  MoveL 4221 to (-399.34, 339.13, -24.94) mm, rotated rx -180 ry 0 rz 0.01 deg; joints [35.63, -31.489, 74.952, -134.207, 54.383, 150.027]
  MoveL 4222 to (-399.69, 339.08, -24.96) mm, rotated rx 180 ry 0 rz 0.01 deg; joints [35.622, -31.473, 74.919, -134.207, 54.368, 150.017]
  MoveL 4223 to (-400.55, 338.85, -24.99) mm, rotated rx 180 ry 0 rz 0.01 deg; joints [35.6, -31.436, 74.847, -134.212, 54.331, 150]
  MoveL 4224 to (-400.6, 338.83, -24.99) mm, rotated rx -180 ry 0 rz 0.01 deg; joints [35.598, -31.435, 74.844, -134.213, 54.329, 149.999]
  MoveL 4225 to (-401.28, 338.49, -25.02) mm, rotated rx -180 ry 0 rz 0.01 deg; joints [35.577, -31.411, 74.798, -134.224, 54.302, 149.993]
  MoveL 4226 to (-401.4, 338.42, -25.02) mm, rotated rx -180 ry 0 rz 0.01 deg; joints [35.572, -31.407, 74.791, -134.227, 54.298, 149.993]
  MoveL 4227 to (-402.84, 337.05, -25.09) mm, rotated rx -180 ry 0 rz 0.01 deg; joints [35.509, -31.38, 74.742, -134.282, 54.25, 150.013]
  MoveL 4228 to (-402.87, 337.02, -25.09) mm, rotated rx 180 ry 0 rz 0.01 deg; joints [35.508, -31.38, 74.742, -134.284, 54.25, 150.014]
  MoveL 4229 to (-403.75, 334.43, -25.19) mm, rotated rx -180 ry 0 rz 0.01 deg; joints [35.423, -31.422, 74.841, -134.402, 54.245, 150.117]
  MoveL 4230 to (-403.78, 333.95, -25.21) mm, rotated rx 180 ry 0 rz 0.01 deg; joints [35.41, -31.437, 74.874, -134.425, 54.251, 150.141]
  MoveL 4231 to (-403.79, 333.65, -25.22) mm, rotated rx 180 ry 0 rz 0.01 deg; joints [35.402, -31.447, 74.895, -134.439, 54.254, 150.156]
  MoveL 4232 to (-403.79, 333.05, -25.24) mm, rotated rx -180 ry 0 rz 0.01 deg; joints [35.386, -31.467, 74.939, -134.468, 54.263, 150.187]
  MoveL 4233 to (-401.25, 328.08, -25.44) mm, rotated rx -180 ry 0 rz 0.01 deg; joints [35.302, -31.758, 75.562, -134.727, 54.453, 150.531]
  MoveL 4234 to (-395.74, 327.2, -25.64) mm, rotated rx 180 ry 0 rz 0.01 deg; joints [35.383, -32.053, 76.188, -134.809, 54.728, 150.769]
  MoveL 4235 to (-391.79, 331.15, -25.85) mm, rotated rx -180 ry 0 rz 0.01 deg; joints [35.562, -32.103, 76.303, -134.652, 54.865, 150.715]
  MoveL 4236 to (-392.66, 336.66, -26.05) mm, rotated rx 180 ry 0 rz 0.01 deg; joints [35.692, -31.86, 75.812, -134.392, 54.757, 150.418]
  MoveL 4237 to (-397.64, 339.2, -26.25) mm, rotated rx -180 ry 0 rz 0.01 deg; joints [35.664, -31.516, 75.116, -134.241, 54.497, 150.126]
  MoveL 4238 to (-398.51, 339.2, -26.28) mm, rotated rx 180 ry 0 rz 0.01 deg; joints [35.648, -31.472, 75.027, -134.236, 54.457, 150.097]
  MoveL 4239 to (-399.34, 339.13, -26.31) mm, rotated rx 180 ry 0 rz 0.01 deg; joints [35.631, -31.431, 74.946, -134.233, 54.42, 150.072]
  MoveL 4240 to (-399.69, 339.08, -26.32) mm, rotated rx 180 ry 0 rz 0.01 deg; joints [35.622, -31.415, 74.913, -134.233, 54.404, 150.063]
  MoveL 4241 to (-400.55, 338.85, -26.35) mm, rotated rx 180 ry 0 rz 0.01 deg; joints [35.6, -31.379, 74.841, -134.238, 54.368, 150.045]
  MoveL 4242 to (-400.6, 338.83, -26.35) mm, rotated rx 180 ry 0 rz 0.01 deg; joints [35.599, -31.377, 74.838, -134.239, 54.366, 150.045]
  MoveL 4243 to (-401.28, 338.49, -26.38) mm, rotated rx -180 ry 0 rz 0.01 deg; joints [35.577, -31.353, 74.792, -134.25, 54.339, 150.038]
  MoveL 4244 to (-401.4, 338.42, -26.39) mm, rotated rx 180 ry 0 rz 0.01 deg; joints [35.573, -31.35, 74.785, -134.253, 54.334, 150.038]
  MoveL 4245 to (-402.84, 337.05, -26.46) mm, rotated rx -180 ry 0 rz 0.01 deg; joints [35.51, -31.322, 74.737, -134.308, 54.287, 150.059]
  MoveL 4246 to (-402.87, 337.02, -26.46) mm, rotated rx -180 ry 0 rz 0.01 deg; joints [35.509, -31.322, 74.737, -134.31, 54.286, 150.06]
  MoveL 4247 to (-403.75, 334.43, -26.55) mm, rotated rx 180 ry 0 rz 0.01 deg; joints [35.424, -31.364, 74.835, -134.428, 54.282, 150.162]
  MoveL 4248 to (-403.78, 333.95, -26.57) mm, rotated rx -180 ry 0 rz 0.01 deg; joints [35.411, -31.379, 74.868, -134.451, 54.287, 150.186]
  MoveL 4249 to (-403.79, 333.65, -26.58) mm, rotated rx 180 ry 0 rz 0.01 deg; joints [35.403, -31.389, 74.889, -134.465, 54.291, 150.201]
  MoveL 4250 to (-403.79, 333.05, -26.6) mm, rotated rx -180 ry 0 rz 0.01 deg; joints [35.387, -31.409, 74.933, -134.494, 54.3, 150.232]
  MoveL 4251 to (-401.25, 328.08, -26.8) mm, rotated rx 180 ry 0 rz 0.01 deg; joints [35.303, -31.7, 75.556, -134.752, 54.49, 150.576]
  MoveL 4252 to (-395.74, 327.2, -27.01) mm, rotated rx -180 ry 0 rz 0.01 deg; joints [35.384, -31.994, 76.182, -134.834, 54.765, 150.814]
  MoveL 4253 to (-391.79, 331.15, -27.21) mm, rotated rx 180 ry 0 rz 0.01 deg; joints [35.563, -32.044, 76.297, -134.678, 54.902, 150.76]
  MoveL 4254 to (-392.66, 336.66, -27.41) mm, rotated rx 180 ry 0 rz 0.01 deg; joints [35.692, -31.802, 75.806, -134.417, 54.794, 150.464]
  MoveL 4255 to (-397.64, 339.2, -27.61) mm, rotated rx -180 ry 0 rz 0.01 deg; joints [35.665, -31.458, 75.11, -134.267, 54.533, 150.172]
  MoveL 4256 to (-398.51, 339.2, -27.64) mm, rotated rx -180 ry 0 rz 0.01 deg; joints [35.649, -31.414, 75.021, -134.262, 54.494, 150.142]
  MoveL 4257 to (-399.34, 339.13, -27.67) mm, rotated rx -180 ry 0 rz 0.01 deg; joints [35.631, -31.373, 74.94, -134.259, 54.456, 150.117]
  MoveL 4258 to (-399.69, 339.08, -27.69) mm, rotated rx -180 ry 0 rz 0.01 deg; joints [35.623, -31.357, 74.907, -134.259, 54.441, 150.108]
  MoveL 4259 to (-400.55, 338.85, -27.72) mm, rotated rx 180 ry 0 rz 0.01 deg; joints [35.601, -31.321, 74.835, -134.265, 54.404, 150.091]
  MoveL 4260 to (-400.6, 338.83, -27.72) mm, rotated rx -180 ry 0 rz 0.01 deg; joints [35.6, -31.319, 74.832, -134.265, 54.403, 150.09]
  MoveL 4261 to (-401.28, 338.49, -27.75) mm, rotated rx -180 ry 0 rz 0.01 deg; joints [35.578, -31.295, 74.786, -134.276, 54.376, 150.084]
  MoveL 4262 to (-401.4, 338.42, -27.75) mm, rotated rx 180 ry 0 rz 0.01 deg; joints [35.574, -31.292, 74.779, -134.279, 54.371, 150.084]
  MoveL 4263 to (-402.84, 337.05, -27.82) mm, rotated rx -180 ry 0 rz 0.01 deg; joints [35.511, -31.264, 74.731, -134.334, 54.323, 150.104]
  MoveL 4264 to (-402.87, 337.02, -27.82) mm, rotated rx -180 ry 0 rz 0.01 deg; joints [35.509, -31.264, 74.731, -134.336, 54.323, 150.105]
  MoveL 4265 to (-403.75, 334.43, -27.92) mm, rotated rx -180 ry 0 rz 0.01 deg; joints [35.424, -31.307, 74.829, -134.454, 54.318, 150.208]
  MoveL 4266 to (-403.78, 333.95, -27.94) mm, rotated rx -180 ry 0 rz 0.01 deg; joints [35.411, -31.321, 74.862, -134.477, 54.324, 150.232]
  MoveL 4267 to (-403.79, 333.65, -27.95) mm, rotated rx -180 ry 0 rz 0.01 deg; joints [35.403, -31.331, 74.883, -134.491, 54.328, 150.246]
  MoveL 4268 to (-403.79, 333.05, -27.97) mm, rotated rx -180 ry 0 rz 0.01 deg; joints [35.387, -31.351, 74.927, -134.52, 54.336, 150.277]
  MoveL 4269 to (-401.25, 328.08, -28.17) mm, rotated rx -180 ry 0 rz 0.01 deg; joints [35.304, -31.642, 75.55, -134.778, 54.527, 150.621]
  MoveL 4270 to (-395.74, 327.2, -28.37) mm, rotated rx -180 ry 0 rz 0.01 deg; joints [35.384, -31.936, 76.176, -134.86, 54.802, 150.859]
  MoveL 4271 to (-391.79, 331.15, -28.57) mm, rotated rx -180 ry 0 rz 0.01 deg; joints [35.564, -31.986, 76.291, -134.703, 54.939, 150.805]
  MoveL 4272 to (-392.66, 336.66, -28.78) mm, rotated rx -180 ry 0 rz 0.01 deg; joints [35.693, -31.744, 75.8, -134.443, 54.831, 150.509]
  MoveL 4273 to (-397.64, 339.2, -28.98) mm, rotated rx -180 ry 0 rz 0.01 deg; joints [35.666, -31.4, 75.104, -134.293, 54.57, 150.217]
  MoveL 4274 to (-398.51, 339.2, -29.01) mm, rotated rx -180 ry 0 rz 0.01 deg; joints [35.649, -31.356, 75.014, -134.287, 54.53, 150.188]
  MoveL 4275 to (-399.34, 339.13, -29.04) mm, rotated rx -180 ry 0 rz 0.01 deg; joints [35.632, -31.315, 74.934, -134.285, 54.493, 150.163]
  MoveL 4276 to (-399.69, 339.08, -29.05) mm, rotated rx -180 ry 0 rz 0.01 deg; joints [35.624, -31.299, 74.901, -134.285, 54.477, 150.154]
  MoveL 4277 to (-400.55, 338.85, -29.08) mm, rotated rx -180 ry 0 rz 0.01 deg; joints [35.601, -31.263, 74.829, -134.29, 54.441, 150.136]
  MoveL 4278 to (-400.6, 338.83, -29.08) mm, rotated rx -180 ry 0 rz 0.01 deg; joints [35.6, -31.261, 74.826, -134.291, 54.439, 150.135]
  MoveL 4279 to (-401.28, 338.49, -29.11) mm, rotated rx 180 ry 0 rz 0.01 deg; joints [35.578, -31.237, 74.78, -134.302, 54.412, 150.129]
  MoveL 4280 to (-401.4, 338.42, -29.12) mm, rotated rx 180 ry 0 rz 0.01 deg; joints [35.574, -31.234, 74.773, -134.305, 54.407, 150.129]
  MoveL 4281 to (-402.84, 337.05, -29.19) mm, rotated rx -180 ry 0 rz 0.01 deg; joints [35.511, -31.206, 74.724, -134.36, 54.36, 150.149]
  MoveL 4282 to (-402.87, 337.02, -29.19) mm, rotated rx -180 ry 0 rz 0.01 deg; joints [35.51, -31.206, 74.724, -134.362, 54.359, 150.15]
  MoveL 4283 to (-403.75, 334.43, -29.28) mm, rotated rx 180 ry 0 rz 0.01 deg; joints [35.425, -31.248, 74.823, -134.48, 54.355, 150.253]
  MoveL 4284 to (-403.78, 333.95, -29.3) mm, rotated rx -180 ry 0 rz 0.01 deg; joints [35.412, -31.263, 74.856, -134.503, 54.361, 150.277]
  MoveL 4285 to (-403.79, 333.65, -29.31) mm, rotated rx -180 ry 0 rz 0.01 deg; joints [35.404, -31.273, 74.876, -134.517, 54.365, 150.292]
  MoveL 4286 to (-403.79, 333.05, -29.33) mm, rotated rx -180 ry 0 rz 0.01 deg; joints [35.388, -31.293, 74.921, -134.546, 54.373, 150.323]
  MoveL 4287 to (-401.25, 328.08, -29.53) mm, rotated rx -180 ry 0 rz 0.01 deg; joints [35.304, -31.583, 75.544, -134.804, 54.564, 150.666]
  MoveL 4288 to (-395.74, 327.2, -29.74) mm, rotated rx -180 ry 0 rz 0.01 deg; joints [35.385, -31.877, 76.17, -134.885, 54.839, 150.904]
  MoveL 4289 to (-391.79, 331.15, -29.94) mm, rotated rx -180 ry 0 rz 0.01 deg; joints [35.564, -31.927, 76.285, -134.729, 54.976, 150.85]
  MoveL 4290 to (-392.66, 336.66, -30.14) mm, rotated rx -180 ry 0 rz 0.01 deg; joints [35.693, -31.685, 75.794, -134.469, 54.867, 150.554]
  MoveL 4291 to (-397.64, 339.2, -30.34) mm, rotated rx -180 ry 0 rz 0.01 deg; joints [35.666, -31.342, 75.098, -134.319, 54.607, 150.262]
  MoveL 4292 to (-398.51, 339.2, -30.37) mm, rotated rx -180 ry 0 rz 0.01 deg; joints [35.65, -31.297, 75.008, -134.313, 54.567, 150.233]
  MoveL 4293 to (-399.34, 339.13, -30.4) mm, rotated rx -180 ry 0 rz 0.01 deg; joints [35.632, -31.257, 74.927, -134.311, 54.529, 150.208]
  MoveL 4294 to (-399.69, 339.08, -30.42) mm, rotated rx -180 ry 0 rz 0.01 deg; joints [35.624, -31.241, 74.895, -134.311, 54.514, 150.199]
  MoveL 4295 to (-400.55, 338.85, -30.45) mm, rotated rx 180 ry 0 rz 0.01 deg; joints [35.602, -31.204, 74.823, -134.316, 54.477, 150.181]
  MoveL 4296 to (-400.6, 338.83, -30.45) mm, rotated rx 180 ry 0 rz 0.01 deg; joints [35.601, -31.203, 74.819, -134.317, 54.475, 150.18]
  MoveL 4297 to (-401.28, 338.49, -30.47) mm, rotated rx -180 ry 0 rz 0.01 deg; joints [35.579, -31.179, 74.773, -134.328, 54.449, 150.174]
  MoveL 4298 to (-401.4, 338.42, -30.48) mm, rotated rx -180 ry 0 rz 0.01 deg; joints [35.575, -31.175, 74.766, -134.331, 54.444, 150.174]
  MoveL 4299 to (-402.84, 337.05, -30.55) mm, rotated rx -180 ry 0 rz 0.01 deg; joints [35.512, -31.148, 74.718, -134.386, 54.396, 150.194]
  MoveL 4300 to (-402.87, 337.02, -30.55) mm, rotated rx -180 ry 0 rz 0.01 deg; joints [35.51, -31.148, 74.718, -134.388, 54.396, 150.195]
  MoveL 4301 to (-403.75, 334.43, -30.65) mm, rotated rx -180 ry 0 rz 0.01 deg; joints [35.426, -31.19, 74.816, -134.506, 54.391, 150.298]
  MoveL 4302 to (-403.78, 333.95, -30.66) mm, rotated rx 180 ry 0 rz 0.01 deg; joints [35.412, -31.205, 74.849, -134.529, 54.397, 150.322]
  MoveL 4303 to (-403.79, 333.65, -30.68) mm, rotated rx -180 ry 0 rz 0.01 deg; joints [35.405, -31.215, 74.87, -134.543, 54.401, 150.337]
  MoveL 4304 to (-403.79, 333.05, -30.7) mm, rotated rx -180 ry 0 rz 0.01 deg; joints [35.389, -31.235, 74.914, -134.572, 54.41, 150.368]
  MoveL 4305 to (-401.25, 328.08, -30.9) mm, rotated rx 180 ry 0 rz 0.01 deg; joints [35.305, -31.525, 75.538, -134.83, 54.601, 150.711]
  MoveL 4306 to (-395.74, 327.2, -31.1) mm, rotated rx 180 ry 0 rz 0.01 deg; joints [35.385, -31.819, 76.164, -134.911, 54.876, 150.949]
  MoveL 4307 to (-391.79, 331.15, -31.3) mm, rotated rx -180 ry 0 rz 0.01 deg; joints [35.565, -31.869, 76.278, -134.754, 55.013, 150.895]
  MoveL 4308 to (-392.66, 336.66, -31.51) mm, rotated rx 180 ry 0 rz 0.01 deg; joints [35.694, -31.627, 75.787, -134.494, 54.904, 150.599]
  MoveL 4309 to (-397.64, 339.2, -31.71) mm, rotated rx -180 ry 0 rz 0.01 deg; joints [35.667, -31.284, 75.091, -134.345, 54.643, 150.307]
  MoveL 4310 to (-398.51, 339.2, -31.74) mm, rotated rx 180 ry 0 rz 0.01 deg; joints [35.65, -31.239, 75.002, -134.339, 54.603, 150.278]
  MoveL 4311 to (-399.34, 339.13, -31.77) mm, rotated rx 180 ry 0 rz 0.01 deg; joints [35.633, -31.199, 74.921, -134.337, 54.566, 150.253]
  MoveL 4312 to (-399.69, 339.08, -31.78) mm, rotated rx -180 ry 0 rz 0.01 deg; joints [35.625, -31.183, 74.888, -134.337, 54.55, 150.244]
  MoveL 4313 to (-400.55, 338.85, -31.81) mm, rotated rx -180 ry 0 rz 0.01 deg; joints [35.603, -31.146, 74.816, -134.342, 54.514, 150.226]
  MoveL 4314 to (-400.6, 338.83, -31.81) mm, rotated rx -180 ry 0 rz 0.01 deg; joints [35.601, -31.145, 74.813, -134.343, 54.512, 150.225]
  MoveL 4315 to (-401.28, 338.49, -31.84) mm, rotated rx 180 ry 0 rz 0.01 deg; joints [35.58, -31.121, 74.767, -134.354, 54.485, 150.219]
  MoveL 4316 to (-401.4, 338.42, -31.84) mm, rotated rx -180 ry 0 rz 0.01 deg; joints [35.575, -31.117, 74.76, -134.357, 54.48, 150.219]
  MoveL 4317 to (-402.84, 337.05, -31.91) mm, rotated rx -180 ry 0 rz 0.01 deg; joints [35.512, -31.09, 74.711, -134.412, 54.433, 150.239]
  MoveL 4318 to (-402.87, 337.02, -31.92) mm, rotated rx -180 ry 0 rz 0.01 deg; joints [35.511, -31.09, 74.711, -134.414, 54.432, 150.24]
  MoveL 4319 to (-403.75, 334.43, -32.01) mm, rotated rx -180 ry 0 rz 0.01 deg; joints [35.426, -31.132, 74.81, -134.532, 54.428, 150.343]
  MoveL 4320 to (-403.78, 333.95, -32.03) mm, rotated rx -180 ry 0 rz 0.01 deg; joints [35.413, -31.147, 74.843, -134.555, 54.434, 150.367]
  MoveL 4321 to (-403.79, 333.65, -32.04) mm, rotated rx -180 ry 0 rz 0.01 deg; joints [35.405, -31.156, 74.863, -134.569, 54.438, 150.382]
  MoveL 4322 to (-403.79, 333.05, -32.06) mm, rotated rx 180 ry 0 rz 0.01 deg; joints [35.389, -31.177, 74.908, -134.598, 54.446, 150.413]
  MoveL 4323 to (-401.25, 328.08, -32.26) mm, rotated rx 180 ry 0 rz 0.01 deg; joints [35.305, -31.467, 75.531, -134.855, 54.638, 150.756]
  MoveL 4324 to (-395.74, 327.2, -32.47) mm, rotated rx -180 ry 0 rz 0.01 deg; joints [35.386, -31.76, 76.157, -134.936, 54.914, 150.994]
  MoveL 4325 to (-391.79, 331.15, -32.67) mm, rotated rx 180 ry 0 rz 0.01 deg; joints [35.565, -31.81, 76.272, -134.779, 55.05, 150.94]
  MoveL 4326 to (-392.66, 336.66, -32.87) mm, rotated rx -180 ry 0 rz 0.01 deg; joints [35.695, -31.568, 75.781, -134.519, 54.941, 150.644]
  MoveL 4327 to (-397.64, 339.2, -33.07) mm, rotated rx -180 ry 0 rz 0.01 deg; joints [35.667, -31.225, 75.085, -134.37, 54.679, 150.352]
  MoveL 4328 to (-398.51, 339.2, -33.1) mm, rotated rx 180 ry 0 rz 0.01 deg; joints [35.651, -31.181, 74.995, -134.365, 54.639, 150.323]
  MoveL 4329 to (-399.34, 339.13, -33.13) mm, rotated rx -180 ry 0 rz 0.01 deg; joints [35.634, -31.141, 74.914, -134.362, 54.602, 150.298]
  MoveL 4330 to (-399.69, 339.08, -33.14) mm, rotated rx 180 ry 0 rz 0.01 deg; joints [35.625, -31.124, 74.882, -134.363, 54.587, 150.289]
  MoveL 4331 to (-400.55, 338.85, -33.18) mm, rotated rx 180 ry 0 rz 0.01 deg; joints [35.603, -31.088, 74.809, -134.368, 54.55, 150.271]
  MoveL 4332 to (-400.6, 338.83, -33.18) mm, rotated rx -180 ry 0 rz 0.01 deg; joints [35.602, -31.086, 74.806, -134.368, 54.548, 150.27]
  MoveL 4333 to (-401.28, 338.49, -33.2) mm, rotated rx -180 ry 0 rz 0.01 deg; joints [35.58, -31.063, 74.76, -134.38, 54.521, 150.264]
  MoveL 4334 to (-401.4, 338.42, -33.21) mm, rotated rx -180 ry 0 rz 0.01 deg; joints [35.576, -31.059, 74.753, -134.382, 54.517, 150.264]
  MoveL 4335 to (-402.84, 337.05, -33.28) mm, rotated rx 180 ry 0 rz 0.01 deg; joints [35.513, -31.032, 74.705, -134.438, 54.469, 150.284]
  MoveL 4336 to (-402.87, 337.02, -33.28) mm, rotated rx -180 ry 0 rz 0.01 deg; joints [35.512, -31.032, 74.705, -134.439, 54.469, 150.285]
  MoveL 4337 to (-403.75, 334.43, -33.38) mm, rotated rx -180 ry 0 rz 0.01 deg; joints [35.427, -31.074, 74.803, -134.557, 54.464, 150.388]
  MoveL 4338 to (-403.78, 333.95, -33.39) mm, rotated rx -180 ry 0 rz 0.01 deg; joints [35.414, -31.089, 74.836, -134.58, 54.47, 150.411]
  MoveL 4339 to (-403.79, 333.65, -33.4) mm, rotated rx -180 ry 0 rz 0.01 deg; joints [35.406, -31.098, 74.857, -134.594, 54.474, 150.426]
  MoveL 4340 to (-403.79, 333.05, -33.43) mm, rotated rx 180 ry 0 rz 0.01 deg; joints [35.39, -31.118, 74.901, -134.623, 54.483, 150.457]
  MoveL 4341 to (-401.25, 328.08, -33.63) mm, rotated rx -180 ry 0 rz 0.01 deg; joints [35.306, -31.408, 75.525, -134.88, 54.675, 150.8]
  MoveL 4342 to (-395.74, 327.2, -33.83) mm, rotated rx -180 ry 0 rz 0.01 deg; joints [35.387, -31.702, 76.15, -134.961, 54.951, 151.038]
  MoveL 4343 to (-391.79, 331.15, -34.03) mm, rotated rx -180 ry 0 rz 0.01 deg; joints [35.566, -31.751, 76.265, -134.805, 55.087, 150.984]
  MoveL 4344 to (-392.66, 336.66, -34.23) mm, rotated rx 180 ry 0 rz 0.01 deg; joints [35.695, -31.51, 75.774, -134.545, 54.977, 150.689]
  MoveL 4345 to (-397.64, 339.2, -34.44) mm, rotated rx -180 ry 0 rz 0.01 deg; joints [35.668, -31.167, 75.078, -134.396, 54.716, 150.397]
  MoveL 4346 to (-398.51, 339.2, -34.47) mm, rotated rx -180 ry 0 rz 0.01 deg; joints [35.652, -31.122, 74.988, -134.39, 54.676, 150.368]
  MoveL 4347 to (-399.34, 339.13, -34.5) mm, rotated rx 180 ry 0 rz 0.01 deg; joints [35.634, -31.082, 74.907, -134.388, 54.639, 150.343]
  MoveL 4348 to (-399.69, 339.08, -34.51) mm, rotated rx -180 ry 0 rz 0.01 deg; joints [35.626, -31.066, 74.875, -134.388, 54.623, 150.334]
  MoveL 4349 to (-400.55, 338.85, -34.54) mm, rotated rx 180 ry 0 rz 0.01 deg; joints [35.604, -31.03, 74.803, -134.393, 54.586, 150.316]
  MoveL 4350 to (-400.6, 338.83, -34.54) mm, rotated rx 180 ry 0 rz 0.01 deg; joints [35.603, -31.028, 74.799, -134.394, 54.585, 150.315]
  MoveL 4351 to (-401.28, 338.49, -34.57) mm, rotated rx -180 ry 0 rz 0.01 deg; joints [35.581, -31.004, 74.753, -134.405, 54.558, 150.309]
  MoveL 4352 to (-401.4, 338.42, -34.57) mm, rotated rx -180 ry 0 rz 0.01 deg; joints [35.576, -31.001, 74.746, -134.408, 54.553, 150.309]
  MoveL 4353 to (-402.84, 337.05, -34.64) mm, rotated rx -180 ry 0 rz 0.01 deg; joints [35.514, -30.974, 74.698, -134.463, 54.506, 150.329]
  MoveL 4354 to (-402.87, 337.02, -34.64) mm, rotated rx -180 ry 0 rz 0.01 deg; joints [35.512, -30.974, 74.698, -134.465, 54.505, 150.33]
  MoveL 4355 to (-403.75, 334.43, -34.74) mm, rotated rx -180 ry 0 rz 0.01 deg; joints [35.427, -31.015, 74.796, -134.583, 54.501, 150.432]
  MoveL 4356 to (-403.78, 333.95, -34.76) mm, rotated rx -180 ry 0 rz 0.01 deg; joints [35.414, -31.03, 74.829, -134.606, 54.507, 150.456]
  MoveL 4357 to (-403.79, 333.65, -34.77) mm, rotated rx -180 ry 0 rz 0.01 deg; joints [35.406, -31.04, 74.85, -134.62, 54.511, 150.471]
  MoveL 4358 to (-403.79, 333.05, -34.79) mm, rotated rx -180 ry 0 rz 0.01 deg; joints [35.39, -31.06, 74.894, -134.649, 54.519, 150.502]
  MoveL 4359 to (-401.25, 328.08, -34.99) mm, rotated rx -180 ry 0 rz 0.01 deg; joints [35.307, -31.35, 75.518, -134.906, 54.712, 150.845]
  MoveL 4360 to (-395.74, 327.2, -35.19) mm, rotated rx 180 ry 0 rz 0.01 deg; joints [35.387, -31.643, 76.144, -134.986, 54.988, 151.083]
  MoveL 4361 to (-391.79, 331.15, -35.4) mm, rotated rx 180 ry 0 rz 0.01 deg; joints [35.566, -31.692, 76.258, -134.83, 55.124, 151.029]
  MoveL 4362 to (-392.66, 336.66, -35.6) mm, rotated rx 180 ry 0 rz 0.01 deg; joints [35.696, -31.451, 75.767, -134.57, 55.014, 150.733]
  MoveL 4363 to (-397.64, 339.2, -35.8) mm, rotated rx 180 ry 0 rz 0.01 deg; joints [35.669, -31.108, 75.071, -134.421, 54.752, 150.442]
  MoveL 4364 to (-398.51, 339.2, -35.83) mm, rotated rx -180 ry 0 rz 0.01 deg; joints [35.652, -31.064, 74.981, -134.416, 54.712, 150.412]
  MoveL 4365 to (-399.34, 339.13, -35.86) mm, rotated rx -180 ry 0 rz 0.01 deg; joints [35.635, -31.024, 74.9, -134.413, 54.675, 150.387]
  MoveL 4366 to (-399.69, 339.08, -35.87) mm, rotated rx -180 ry 0 rz 0.01 deg; joints [35.627, -31.007, 74.868, -134.414, 54.659, 150.378]
  MoveL 4367 to (-400.55, 338.85, -35.9) mm, rotated rx -180 ry 0 rz 0.01 deg; joints [35.604, -30.971, 74.796, -134.419, 54.623, 150.361]
  MoveL 4368 to (-400.6, 338.83, -35.91) mm, rotated rx -180 ry 0 rz 0.01 deg; joints [35.603, -30.97, 74.792, -134.419, 54.621, 150.36]
  MoveL 4369 to (-401.28, 338.49, -35.93) mm, rotated rx -180 ry 0 rz 0.01 deg; joints [35.581, -30.946, 74.746, -134.431, 54.594, 150.354]
  MoveL 4370 to (-401.4, 338.42, -35.94) mm, rotated rx -180 ry 0 rz 0.01 deg; joints [35.577, -30.942, 74.739, -134.434, 54.589, 150.353]
  MoveL 4371 to (-402.84, 337.05, -36.01) mm, rotated rx -180 ry 0 rz 0.01 deg; joints [35.514, -30.915, 74.691, -134.489, 54.542, 150.374]
  MoveL 4372 to (-402.87, 337.02, -36.01) mm, rotated rx -180 ry 0 rz 0.01 deg; joints [35.513, -30.915, 74.691, -134.49, 54.541, 150.375]
  MoveL 4373 to (-403.75, 334.43, -36.11) mm, rotated rx -180 ry 0 rz 0.01 deg; joints [35.428, -30.957, 74.789, -134.608, 54.537, 150.477]
  MoveL 4374 to (-403.78, 333.95, -36.12) mm, rotated rx -180 ry 0 rz 0.01 deg; joints [35.415, -30.972, 74.822, -134.631, 54.543, 150.501]
  MoveL 4375 to (-403.79, 333.65, -36.13) mm, rotated rx -180 ry 0 rz 0.01 deg; joints [35.407, -30.981, 74.843, -134.645, 54.547, 150.516]
  MoveL 4376 to (-403.79, 333.05, -36.15) mm, rotated rx -180 ry 0 rz 0.01 deg; joints [35.391, -31.001, 74.887, -134.674, 54.556, 150.546]
  MoveL 4377 to (-401.25, 328.08, -36.36) mm, rotated rx -180 ry 0 rz 0.01 deg; joints [35.307, -31.291, 75.511, -134.931, 54.749, 150.889]
  MoveL 4378 to (-395.74, 327.2, -36.56) mm, rotated rx 180 ry 0 rz 0.01 deg; joints [35.388, -31.584, 76.137, -135.012, 55.025, 151.127]
  MoveL 4379 to (-391.79, 331.15, -36.76) mm, rotated rx -180 ry 0 rz 0.01 deg; joints [35.567, -31.634, 76.251, -134.855, 55.161, 151.073]
  MoveL 4380 to (-392.66, 336.66, -36.96) mm, rotated rx 180 ry 0 rz 0.01 deg; joints [35.696, -31.392, 75.76, -134.595, 55.051, 150.778]
  MoveL 4381 to (-397.64, 339.2, -37.17) mm, rotated rx -180 ry 0 rz 0.01 deg; joints [35.669, -31.05, 75.064, -134.446, 54.788, 150.486]
  MoveL 4382 to (-398.51, 339.2, -37.2) mm, rotated rx -180 ry 0 rz 0.01 deg; joints [35.653, -31.005, 74.974, -134.441, 54.748, 150.457]
  MoveL 4383 to (-399.34, 339.13, -37.23) mm, rotated rx -180 ry 0 rz 0.01 deg; joints [35.635, -30.965, 74.893, -134.439, 54.711, 150.432]
  MoveL 4384 to (-399.69, 339.08, -37.24) mm, rotated rx -180 ry 0 rz 0.01 deg; joints [35.627, -30.949, 74.861, -134.439, 54.695, 150.423]
  MoveL 4385 to (-400.55, 338.85, -37.27) mm, rotated rx 180 ry 0 rz 0.01 deg; joints [35.605, -30.913, 74.788, -134.444, 54.659, 150.405]
  MoveL 4386 to (-400.6, 338.83, -37.27) mm, rotated rx -180 ry 0 rz 0.01 deg; joints [35.604, -30.911, 74.785, -134.445, 54.657, 150.404]
  MoveL 4387 to (-401.28, 338.49, -37.3) mm, rotated rx 180 ry 0 rz 0.01 deg; joints [35.582, -30.888, 74.739, -134.456, 54.63, 150.398]
  MoveL 4388 to (-401.4, 338.42, -37.3) mm, rotated rx -180 ry 0 rz 0.01 deg; joints [35.578, -30.884, 74.732, -134.459, 54.625, 150.398]
  MoveL 4389 to (-402.84, 337.05, -37.37) mm, rotated rx -180 ry 0 rz 0.01 deg; joints [35.515, -30.857, 74.684, -134.514, 54.578, 150.418]
  MoveL 4390 to (-402.87, 337.02, -37.37) mm, rotated rx -180 ry 0 rz 0.01 deg; joints [35.513, -30.857, 74.684, -134.516, 54.578, 150.419]
  MoveL 4391 to (-403.75, 334.43, -37.47) mm, rotated rx 180 ry 0 rz 0.01 deg; joints [35.429, -30.899, 74.782, -134.634, 54.574, 150.521]
  MoveL 4392 to (-403.78, 333.95, -37.49) mm, rotated rx -180 ry 0 rz 0.01 deg; joints [35.415, -30.913, 74.815, -134.657, 54.58, 150.545]
  MoveL 4393 to (-403.79, 333.65, -37.5) mm, rotated rx 180 ry 0 rz 0.01 deg; joints [35.407, -30.923, 74.836, -134.671, 54.583, 150.56]
  MoveL 4394 to (-403.79, 333.05, -37.52) mm, rotated rx 180 ry 0 rz 0.01 deg; joints [35.392, -30.943, 74.88, -134.7, 54.592, 150.591]
  MoveL 4395 to (-401.25, 328.08, -37.72) mm, rotated rx -180 ry 0 rz 0.01 deg; joints [35.308, -31.232, 75.503, -134.956, 54.785, 150.934]
  MoveL 4396 to (-395.74, 327.2, -37.92) mm, rotated rx 180 ry 0 rz 0.01 deg; joints [35.388, -31.525, 76.129, -135.036, 55.061, 151.172]
  MoveL 4397 to (-391.79, 331.15, -38.13) mm, rotated rx -180 ry 0 rz 0.01 deg; joints [35.568, -31.575, 76.244, -134.88, 55.198, 151.118]
  MoveL 4398 to (-392.66, 336.66, -38.33) mm, rotated rx -180 ry 0 rz 0.01 deg; joints [35.697, -31.333, 75.753, -134.62, 55.087, 150.822]
  MoveL 4399 to (-397.64, 339.2, -38.53) mm, rotated rx -180 ry 0 rz 0.01 deg; joints [35.67, -30.991, 75.056, -134.472, 54.825, 150.531]
  MoveL 4400 to (-398.51, 339.2, -38.56) mm, rotated rx -180 ry 0 rz 0.01 deg; joints [35.653, -30.947, 74.967, -134.466, 54.785, 150.501]
  MoveL 4401 to (-399.34, 339.13, -38.59) mm, rotated rx -180 ry 0 rz 0.01 deg; joints [35.636, -30.907, 74.886, -134.464, 54.747, 150.476]
  MoveL 4402 to (-399.69, 339.08, -38.6) mm, rotated rx 180 ry 0 rz 0.01 deg; joints [35.628, -30.89, 74.853, -134.464, 54.732, 150.467]
  MoveL 4403 to (-400.55, 338.85, -38.63) mm, rotated rx 180 ry 0 rz 0.01 deg; joints [35.606, -30.854, 74.781, -134.469, 54.695, 150.45]
  MoveL 4404 to (-400.6, 338.83, -38.64) mm, rotated rx -180 ry 0 rz 0.01 deg; joints [35.604, -30.852, 74.778, -134.47, 54.693, 150.449]
  MoveL 4405 to (-401.28, 338.49, -38.66) mm, rotated rx -180 ry 0 rz 0.01 deg; joints [35.583, -30.829, 74.732, -134.481, 54.666, 150.443]
  MoveL 4406 to (-401.4, 338.42, -38.67) mm, rotated rx -180 ry 0 rz 0.01 deg; joints [35.578, -30.825, 74.725, -134.484, 54.662, 150.442]
  MoveL 4407 to (-402.84, 337.05, -38.74) mm, rotated rx -180 ry 0 rz 0.01 deg; joints [35.515, -30.798, 74.676, -134.54, 54.614, 150.463]
  MoveL 4408 to (-402.87, 337.02, -38.74) mm, rotated rx -180 ry 0 rz 0.01 deg; joints [35.514, -30.798, 74.676, -134.541, 54.614, 150.464]
  MoveL 4409 to (-403.75, 334.43, -38.84) mm, rotated rx -180 ry 0 rz 0.01 deg; joints [35.429, -30.84, 74.775, -134.659, 54.61, 150.566]
  MoveL 4410 to (-403.78, 333.95, -38.85) mm, rotated rx -180 ry 0 rz 0.01 deg; joints [35.416, -30.855, 74.807, -134.682, 54.616, 150.59]
  MoveL 4411 to (-403.79, 333.65, -38.86) mm, rotated rx -180 ry 0 rz 0.01 deg; joints [35.408, -30.864, 74.828, -134.696, 54.62, 150.604]
  MoveL 4412 to (-403.79, 333.05, -38.88) mm, rotated rx -180 ry 0 rz 0.01 deg; joints [35.392, -30.884, 74.872, -134.725, 54.629, 150.635]
  MoveL 4413 to (-401.25, 328.08, -39.09) mm, rotated rx 180 ry 0 rz 0.01 deg; joints [35.308, -31.173, 75.496, -134.981, 54.822, 150.978]
  MoveL 4414 to (-395.74, 327.2, -39.29) mm, rotated rx -180 ry 0 rz 0.01 deg; joints [35.389, -31.466, 76.122, -135.061, 55.098, 151.216]
  MoveL 4415 to (-391.79, 331.15, -39.49) mm, rotated rx -180 ry 0 rz 0.01 deg; joints [35.568, -31.516, 76.236, -134.904, 55.234, 151.162]
  MoveL 4416 to (-392.66, 336.66, -39.69) mm, rotated rx 180 ry 0 rz 0.01 deg; joints [35.698, -31.274, 75.745, -134.645, 55.124, 150.867]
  MoveL 4417 to (-397.64, 339.2, -39.9) mm, rotated rx -180 ry 0 rz 0.01 deg; joints [35.67, -30.932, 75.049, -134.497, 54.861, 150.575]
  MoveL 4418 to (-398.51, 339.2, -39.93) mm, rotated rx -180 ry 0 rz 0.01 deg; joints [35.654, -30.888, 74.959, -134.491, 54.821, 150.546]
  MoveL 4419 to (-399.34, 339.13, -39.95) mm, rotated rx -180 ry 0 rz 0.01 deg; joints [35.637, -30.848, 74.878, -134.489, 54.783, 150.521]
  MoveL 4420 to (-399.69, 339.08, -39.97) mm, rotated rx -180 ry 0 rz 0.01 deg; joints [35.628, -30.832, 74.846, -134.489, 54.768, 150.512]
  MoveL 4421 to (-400.55, 338.85, -40) mm, rotated rx -180 ry 0 rz 0.01 deg; joints [35.606, -30.795, 74.774, -134.495, 54.731, 150.494]
  MoveL 4422 to (-400.6, 338.83, -40) mm, rotated rx -180 ry 0 rz 0.01 deg; joints [35.605, -30.794, 74.77, -134.495, 54.729, 150.493]
  MoveL 4423 to (-400.13, 339.01, -40) mm, rotated rx -180 ry 0 rz 0.01 deg; joints [35.618, -30.811, 74.805, -134.49, 54.749, 150.501]
  MoveL 4424 to (-398.92, 339.2, -40) mm, rotated rx -180 ry 0 rz 0.01 deg; joints [35.646, -30.864, 74.916, -134.49, 54.803, 150.533]
  MoveL 4425 to (-213.35, 339.2, -40) mm, rotated rx 180 ry 0 rz 0.01 deg; joints [39.468, -38.9, 91.717, -134.344, 62.753, 155.77]
  MoveL 4426 to (-213.55, 339.16, -40) mm, rotated rx 180 ry 0 rz 0.01 deg; joints [39.462, -38.894, 91.704, -134.347, 62.746, 155.767]
  MoveL 4427 to (-214.63, 338.89, -40) mm, rotated rx 180 ry 0 rz 0.01 deg; joints [39.43, -38.861, 91.635, -134.366, 62.707, 155.753]
  MoveL 4428 to (-215.28, 338.65, -40) mm, rotated rx 180 ry 0 rz 0.01 deg; joints [39.409, -38.844, 91.598, -134.38, 62.685, 155.748]
  MoveL 4429 to (-225.8, 333.55, -40) mm, rotated rx -180 ry 0 rz 0.01 deg; joints [39.036, -38.596, 91.083, -134.661, 62.336, 155.712]
  MoveL 4430 to (-226.11, 333.38, -40) mm, rotated rx 180 ry 0 rz 0.01 deg; joints [39.024, -38.589, 91.069, -134.67, 62.326, 155.712]
  MoveL 4431 to (-227.57, 332.48, -40) mm, rotated rx 180 ry 0 rz 0.01 deg; joints [38.967, -38.56, 91.01, -134.716, 62.28, 155.715]
  MoveL 4432 to (-228.07, 332.1, -40) mm, rotated rx 180 ry 0 rz 0.01 deg; joints [38.946, -38.553, 90.994, -134.735, 62.265, 155.719]
  MoveL 4433 to (-229.52, 330.77, -40) mm, rotated rx -180 ry 0 rz 0.01 deg; joints [38.877, -38.537, 90.964, -134.799, 62.224, 155.74]
  MoveL 4434 to (-229.56, 330.73, -40) mm, rotated rx 180 ry 0 rz 0.01 deg; joints [38.875, -38.537, 90.963, -134.801, 62.223, 155.741]
  MoveL 4435 to (-236.64, 324.01, -40) mm, rotated rx 180 ry 0 rz 0.01 deg; joints [38.536, -38.466, 90.823, -135.122, 62.028, 155.852]
  MoveL 4436 to (-236.94, 323.69, -40) mm, rotated rx 180 ry 0 rz 0.01 deg; joints [38.52, -38.464, 90.82, -135.137, 62.02, 155.858]
  MoveL 4437 to (-237.82, 322.6, -40) mm, rotated rx -180 ry 0 rz 0.01 deg; joints [38.471, -38.463, 90.818, -135.187, 61.999, 155.882]
  MoveL 4438 to (-238.12, 322.17, -40) mm, rotated rx -180 ry 0 rz 0.01 deg; joints [38.453, -38.464, 90.822, -135.207, 61.993, 155.893]
  MoveL 4439 to (-240.45, 318.18, -40) mm, rotated rx -180 ry 0 rz 0.01 deg; joints [38.292, -38.493, 90.89, -135.386, 61.951, 156.002]
  MoveL 4440 to (-240.49, 318.11, -40) mm, rotated rx 180 ry 0 rz 0.01 deg; joints [38.289, -38.494, 90.891, -135.389, 61.95, 156.005]
  MoveL 4441 to (-243.68, 312.3, -40) mm, rotated rx -180 ry 0 rz 0.01 deg; joints [38.059, -38.544, 91.004, -135.648, 61.897, 156.168]
  MoveL 4442 to (-243.84, 311.95, -40) mm, rotated rx 180 ry 0 rz 0.01 deg; joints [38.046, -38.548, 91.013, -135.663, 61.895, 156.178]
  MoveL 4443 to (-244.73, 309.78, -40) mm, rotated rx 180 ry 0 rz 0.01 deg; joints [37.967, -38.578, 91.08, -135.759, 61.888, 156.247]
  MoveL 4444 to (-244.95, 309.01, -40) mm, rotated rx -180 ry 0 rz 0.01 deg; joints [37.941, -38.592, 91.111, -135.792, 61.889, 156.273]
  MoveL 4445 to (-246.39, 299.58, -40) mm, rotated rx 180 ry 0 rz 0.01 deg; joints [37.647, -38.815, 91.595, -136.19, 61.953, 156.624]
  MoveL 4446 to (-246.42, 299.36, -40) mm, rotated rx 180 ry 0 rz 0.01 deg; joints [37.64, -38.821, 91.607, -136.2, 61.955, 156.632]
  MoveL 4447 to (-246.51, 298.27, -40) mm, rotated rx -180 ry 0 rz 0.01 deg; joints [37.608, -38.849, 91.669, -136.245, 61.965, 156.674]
  MoveC 4448 to (-246.51, 297.75, -40) mm, rotated rx -180 ry 0 rz 0.01 deg; joints [37.593, -38.864, 91.701, -136.267, 61.972, 156.695] to (-246.44, 297.24, -40) mm, rotated rx -180 ry 0 rz 0.01 deg; joints [37.581, -38.882, 91.739, -136.287, 61.981, 156.718]
  MoveL 4449 to (-245.04, 290.98, -40) mm, rotated rx 180 ry 0 rz 0.01 deg; joints [37.435, -39.119, 92.249, -136.537, 62.118, 157.002]
  MoveL 4450 to (-245.03, 290.91, -40) mm, rotated rx 180 ry 0 rz 0.01 deg; joints [37.434, -39.122, 92.255, -136.54, 62.12, 157.005]
  MoveL 4451 to (-244.07, 287.02, -40) mm, rotated rx 180 ry 0 rz 0.01 deg; joints [37.344, -39.272, 92.578, -136.694, 62.209, 157.183]
  MoveL 4452 to (-243.75, 286.18, -40) mm, rotated rx 180 ry 0 rz 0.01 deg; joints [37.328, -39.308, 92.656, -136.726, 62.232, 157.224]
  MoveL 4453 to (-241.42, 281.98, -40) mm, rotated rx -180 ry 0 rz 0.01 deg; joints [37.259, -39.519, 93.108, -136.884, 62.38, 157.444]
  MoveL 4454 to (-241.22, 281.66, -40) mm, rotated rx -180 ry 0 rz 0.01 deg; joints [37.254, -39.536, 93.144, -136.896, 62.392, 157.461]
  MoveL 4455 to (-240.29, 280.35, -40) mm, rotated rx 180 ry 0 rz 0.01 deg; joints [37.237, -39.609, 93.301, -136.943, 62.446, 157.534]
  MoveL 4456 to (-240.11, 280.11, -40) mm, rotated rx -180 ry 0 rz 0.01 deg; joints [37.234, -39.623, 93.331, -136.952, 62.457, 157.548]
  MoveL 4457 to (-237.06, 276.55, -40) mm, rotated rx 180 ry 0 rz 0.01 deg; joints [37.199, -39.842, 93.798, -137.077, 62.625, 157.756]
  MoveL 4458 to (-236.75, 276.23, -40) mm, rotated rx 180 ry 0 rz 0.01 deg; joints [37.197, -39.863, 93.844, -137.087, 62.641, 157.776]
  MoveL 4459 to (-236.39, 275.91, -40) mm, rotated rx 180 ry 0 rz 0.01 deg; joints [37.195, -39.886, 93.893, -137.098, 62.66, 157.797]
  MoveL 4460 to (-236.12, 275.69, -40) mm, rotated rx -180 ry 0 rz 0.01 deg; joints [37.195, -39.903, 93.928, -137.105, 62.674, 157.811]
  MoveL 4461 to (-230.67, 271.73, -40) mm, rotated rx -180 ry 0 rz 0.01 deg; joints [37.2, -40.222, 94.611, -137.227, 62.942, 158.086]
  MoveL 4462 to (-230.2, 271.44, -40) mm, rotated rx 180 ry 0 rz 0.01 deg; joints [37.202, -40.248, 94.667, -137.235, 62.965, 158.108]
  MoveL 4463 to (-227.17, 269.92, -40) mm, rotated rx -180 ry 0 rz 0.01 deg; joints [37.224, -40.406, 95.003, -137.274, 63.104, 158.233]
  MoveL 4464 to (-226.74, 269.75, -40) mm, rotated rx 180 ry 0 rz 0.01 deg; joints [37.228, -40.427, 95.048, -137.277, 63.124, 158.249]
  MoveL 4465 to (-223.24, 268.55, -40) mm, rotated rx 180 ry 0 rz 0.01 deg; joints [37.271, -40.592, 95.401, -137.298, 63.278, 158.371]
  MoveL 4466 to (-222.62, 268.41, -40) mm, rotated rx -180 ry 0 rz 0.01 deg; joints [37.28, -40.62, 95.459, -137.299, 63.304, 158.391]
  MoveL 4467 to (-215.36, 267.4, -40) mm, rotated rx -180 ry 0 rz 0.01 deg; joints [37.41, -40.92, 96.098, -137.279, 63.603, 158.586]
  MoveL 4468 to (-214.9, 267.36, -40) mm, rotated rx -180 ry 0 rz 0.01 deg; joints [37.42, -40.939, 96.136, -137.277, 63.622, 158.597]
  MoveL 4469 to (-178.62, 267.36, -40) mm, rotated rx -180 ry 0 rz 0.01 deg; joints [38.234, -42.265, 98.956, -136.93, 65.027, 159.354]
  MoveL 4470 to (-178.15, 267.4, -40) mm, rotated rx -180 ry 0 rz 0.01 deg; joints [38.246, -42.28, 98.99, -136.924, 65.044, 159.362]
  MoveL 4471 to (-170.89, 268.41, -40) mm, rotated rx 180 ry 0 rz 0.01 deg; joints [38.442, -42.511, 99.481, -136.806, 65.307, 159.472]
  MoveL 4472 to (-170.31, 268.54, -40) mm, rotated rx 180 ry 0 rz 0.01 deg; joints [38.459, -42.528, 99.517, -136.794, 65.327, 159.479]
  MoveL 4473 to (-167.48, 269.46, -40) mm, rotated rx -180 ry 0 rz 0.01 deg; joints [38.551, -42.604, 99.676, -136.726, 65.423, 159.502]
  MoveL 4474 to (-167.1, 269.61, -40) mm, rotated rx -180 ry 0 rz 0.01 deg; joints [38.564, -42.613, 99.695, -136.716, 65.435, 159.504]
  MoveL 4475 to (-164.14, 270.98, -40) mm, rotated rx 180 ry 0 rz 0.01 deg; joints [38.673, -42.68, 99.836, -136.629, 65.529, 159.512]
  MoveL 4476 to (-163.71, 271.21, -40) mm, rotated rx -180 ry 0 rz 0.01 deg; joints [38.689, -42.688, 99.854, -136.614, 65.542, 159.512]
  MoveL 4477 to (-161.53, 272.63, -40) mm, rotated rx 180 ry 0 rz 0.01 deg; joints [38.781, -42.726, 99.932, -136.534, 65.606, 159.503]
  MoveL 4478 to (-161.34, 272.76, -40) mm, rotated rx 180 ry 0 rz 0.01 deg; joints [38.79, -42.729, 99.939, -136.526, 65.611, 159.502]
  MoveL 4479 to (-156.98, 276.05, -40) mm, rotated rx -180 ry 0 rz 0.01 deg; joints [38.987, -42.792, 100.067, -136.346, 65.733, 159.467]
  MoveL 4480 to (-156.45, 276.55, -40) mm, rotated rx -180 ry 0 rz 0.01 deg; joints [39.014, -42.797, 100.077, -136.32, 65.746, 159.459]
  MoveL 4481 to (-153.97, 279.45, -40) mm, rotated rx -180 ry 0 rz 0.01 deg; joints [39.156, -42.803, 100.086, -136.176, 65.801, 159.4]
  MoveL 4482 to (-153.84, 279.61, -40) mm, rotated rx 180 ry 0 rz 0.01 deg; joints [39.163, -42.803, 100.086, -136.169, 65.804, 159.397]
  MoveL 4483 to (-152.35, 281.58, -40) mm, rotated rx -180 ry 0 rz 0.01 deg; joints [39.255, -42.801, 100.078, -136.074, 65.834, 159.353]
  MoveL 4484 to (-152.09, 281.98, -40) mm, rotated rx 180 ry 0 rz 0.01 deg; joints [39.273, -42.799, 100.073, -136.055, 65.839, 159.343]
  MoveL 4485 to (-149.77, 286.18, -40) mm, rotated rx -180 ry 0 rz 0.01 deg; joints [39.449, -42.763, 99.989, -135.861, 65.871, 159.232]
  MoveL 4486 to (-149.43, 287.04, -40) mm, rotated rx -180 ry 0 rz 0.01 deg; joints [39.481, -42.751, 99.962, -135.824, 65.872, 159.207]
  MoveL 4487 to (-147.12, 296.84, -40) mm, rotated rx 180 ry 0 rz 0.01 deg; joints [39.816, -42.556, 99.532, -135.41, 65.831, 158.884]
  MoveL 4488 to (-147.03, 297.46, -40) mm, rotated rx -180 ry 0 rz 0.01 deg; joints [39.836, -42.542, 99.5, -135.385, 65.826, 158.862]
  MoveL 4489 to (-146.99, 298.18, -40) mm, rotated rx 180 ry 0 rz 0.01 deg; joints [39.857, -42.522, 99.457, -135.356, 65.818, 158.835]
  MoveL 4490 to (-147.03, 298.84, -40) mm, rotated rx 180 ry 0 rz 0.01 deg; joints [39.875, -42.503, 99.414, -135.33, 65.808, 158.81]
  MoveL 4491 to (-148.48, 308.63, -40) mm, rotated rx 180 ry 0 rz 0.01 deg; joints [40.118, -42.172, 98.696, -134.961, 65.627, 158.405]
  MoveL 4492 to (-148.63, 309.24, -40) mm, rotated rx 180 ry 0 rz 0.01 deg; joints [40.132, -42.15, 98.647, -134.939, 65.613, 158.379]
  MoveL 4493 to (-149.26, 311.05, -40) mm, rotated rx 180 ry 0 rz 0.01 deg; joints [40.168, -42.076, 98.486, -134.874, 65.567, 158.296]
  MoveL 4494 to (-149.46, 311.52, -40) mm, rotated rx 180 ry 0 rz 0.01 deg; joints [40.176, -42.055, 98.441, -134.858, 65.553, 158.274]
  MoveL 4495 to (-151.37, 315.15, -40) mm, rotated rx -180 ry 0 rz 0.01 deg; joints [40.233, -41.883, 98.07, -134.736, 65.435, 158.094]
  MoveL 4496 to (-151.42, 315.25, -40) mm, rotated rx -180 ry 0 rz 0.01 deg; joints [40.234, -41.879, 98.06, -134.733, 65.432, 158.089]
  MoveL 4497 to (-155.13, 321.78, -40) mm, rotated rx 180 ry 0 rz 0.01 deg; joints [40.329, -41.558, 97.368, -134.516, 65.208, 157.758]
  MoveL 4498 to (-155.37, 322.14, -40) mm, rotated rx 180 ry 0 rz 0.01 deg; joints [40.333, -41.539, 97.327, -134.504, 65.195, 157.738]
  MoveL 4499 to (-156.19, 323.23, -40) mm, rotated rx -180 ry 0 rz 0.01 deg; joints [40.344, -41.478, 97.196, -134.47, 65.15, 157.678]
  MoveL 4500 to (-156.47, 323.55, -40) mm, rotated rx 180 ry 0 rz 0.01 deg; joints [40.347, -41.458, 97.154, -134.46, 65.135, 157.66]
  MoveL 4501 to (-157.53, 324.64, -40) mm, rotated rx 180 ry 0 rz 0.01 deg; joints [40.352, -41.389, 97.005, -134.429, 65.081, 157.595]
  MoveL 4502 to (-157.63, 324.74, -40) mm, rotated rx 180 ry 0 rz 0.01 deg; joints [40.352, -41.382, 96.991, -134.426, 65.076, 157.589]
  MoveL 4503 to (-165.05, 331.75, -40) mm, rotated rx 180 ry 0 rz 0.01 deg; joints [40.372, -40.91, 95.979, -134.225, 64.707, 157.153]
  MoveL 4504 to (-165.4, 332.04, -40) mm, rotated rx 180 ry 0 rz 0.01 deg; joints [40.372, -40.889, 95.933, -134.217, 64.69, 157.134]
  MoveL 4505 to (-166.85, 333.08, -40) mm, rotated rx 180 ry 0 rz 0.01 deg; joints [40.366, -40.806, 95.755, -134.19, 64.622, 157.062]
  MoveL 4506 to (-167.34, 333.37, -40) mm, rotated rx -180 ry 0 rz 0.01 deg; joints [40.363, -40.78, 95.699, -134.184, 64.599, 157.039]
  MoveL 4507 to (-177.86, 338.5, -40) mm, rotated rx 180 ry 0 rz 0.01 deg; joints [40.258, -40.245, 94.558, -134.08, 64.134, 156.604]
  MoveL 4508 to (-178.19, 338.64, -40) mm, rotated rx -180 ry 0 rz 0.01 deg; joints [40.255, -40.228, 94.524, -134.078, 64.12, 156.591]
  MoveL 4509 to (-178.91, 338.9, -40) mm, rotated rx 180 ry 0 rz 0.01 deg; joints [40.245, -40.194, 94.451, -134.074, 64.089, 156.564]
  MoveL 4510 to (-179.55, 339.06, -40) mm, rotated rx 180 ry 0 rz 0.01 deg; joints [40.235, -40.166, 94.391, -134.073, 64.062, 156.543]
  MoveL 4511 to (-180.46, 339.2, -40) mm, rotated rx 180 ry 0 rz 0.01 deg; joints [40.218, -40.128, 94.311, -134.076, 64.026, 156.518]
  MoveL 4512 to (4.87, 339.21, -40) mm, rotated rx -180 ry 0 rz 0.01 deg; joints [44.916, -46.237, 107.372, -131.517, 70.593, 160.189]
  MoveL 4513 to (5.94, 339.15, -40) mm, rotated rx -180 ry 0 rz 0.01 deg; joints [44.944, -46.27, 107.444, -131.5, 70.629, 160.211]
  MoveL 4514 to (6.8, 338.95, -40) mm, rotated rx 180 ry 0 rz 0.01 deg; joints [44.963, -46.301, 107.512, -131.491, 70.66, 160.233]
  MoveL 4515 to (7.07, 338.84, -40) mm, rotated rx 180 ry 0 rz 0.01 deg; joints [44.967, -46.313, 107.537, -131.49, 70.671, 160.243]
  MoveL 4516 to (7.37, 338.63, -40) mm, rotated rx 180 ry 0 rz 0.01 deg; joints [44.97, -46.328, 107.569, -131.492, 70.683, 160.256]
  MoveL 4517 to (9.66, 336.38, -40) mm, rotated rx -180 ry 0 rz 0.01 deg; joints [44.971, -46.46, 107.86, -131.533, 70.788, 160.381]
  MoveL 4518 to (9.9, 336.02, -40) mm, rotated rx 180 ry 0 rz 0.01 deg; joints [44.967, -46.477, 107.898, -131.542, 70.801, 160.398]
  MoveL 4519 to (10.07, 335.56, -40) mm, rotated rx -180 ry 0 rz 0.01 deg; joints [44.959, -46.496, 107.938, -131.555, 70.813, 160.418]
  MoveL 4520 to (10.27, 334.35, -40) mm, rotated rx -180 ry 0 rz 0.01 deg; joints [44.931, -46.536, 108.028, -131.596, 70.835, 160.467]
  MoveL 4521 to (10.27, 31.87, -40) mm, rotated rx 180 ry 0 rz 0.01 deg; joints [35.133, -53.75, 124.619, -143.431, 75.064, 170.12]
  MoveL 4522 to (9.18, 36.46, -40) mm, rotated rx 180 ry 0 rz 0.01 deg; joints [35.275, -53.63, 124.332, -143.261, 74.958, 169.978]
  MoveL 4523 to (9.03, 36.92, -40) mm, rotated rx 180 ry 0 rz 0.01 deg; joints [35.288, -53.617, 124.301, -143.244, 74.947, 169.963]
  MoveL 4524 to (8.48, 38.3, -40) mm, rotated rx 180 ry 0 rz 0.01 deg; joints [35.325, -53.574, 124.201, -143.198, 74.908, 169.918]
  MoveL 4525 to (8.27, 38.74, -40) mm, rotated rx 180 ry 0 rz 0.01 deg; joints [35.336, -53.559, 124.166, -143.184, 74.894, 169.902]
  MoveL 4526 to (6.11, 42.48, -40) mm, rotated rx 180 ry 0 rz 0.01 deg; joints [35.417, -53.424, 123.848, -143.071, 74.764, 169.766]
  MoveL 4527 to (6.07, 42.54, -40) mm, rotated rx -180 ry 0 rz 0.01 deg; joints [35.418, -53.422, 123.843, -143.069, 74.762, 169.764]
  MoveL 4528 to (2.56, 48.35, -40) mm, rotated rx -180 ry 0 rz 0.01 deg; joints [35.539, -53.206, 123.337, -142.899, 74.555, 169.549]
  MoveL 4529 to (2.35, 48.65, -40) mm, rotated rx 180 ry 0 rz 0.01 deg; joints [35.545, -53.193, 123.308, -142.89, 74.543, 169.537]
  MoveL 4530 to (1.05, 50.35, -40) mm, rotated rx 180 ry 0 rz 0.01 deg; joints [35.573, -53.122, 123.142, -142.846, 74.473, 169.47]
  MoveL 4531 to (0.48, 50.92, -40) mm, rotated rx 180 ry 0 rz 0.01 deg; joints [35.579, -53.094, 123.077, -142.833, 74.445, 169.445]
  MoveL 4532 to (-7.44, 57.29, -40) mm, rotated rx -180 ry 0 rz 0.01 deg; joints [35.605, -52.736, 122.248, -142.727, 74.076, 169.142]
  MoveL 4533 to (-7.81, 57.56, -40) mm, rotated rx 180 ry 0 rz 0.01 deg; joints [35.605, -52.72, 122.211, -142.724, 74.059, 169.129]
  MoveL 4534 to (-8.47, 57.96, -40) mm, rotated rx 180 ry 0 rz 0.01 deg; joints [35.602, -52.692, 122.148, -142.72, 74.03, 169.107]
  MoveL 4535 to (-9.24, 58.3, -40) mm, rotated rx -180 ry 0 rz 0.01 deg; joints [35.594, -52.663, 122.08, -142.721, 73.998, 169.085]
  MoveL 4536 to (-19.1, 61.28, -40) mm, rotated rx 180 ry 0 rz 0.01 deg; joints [35.448, -52.311, 121.279, -142.791, 73.608, 168.845]
  MoveL 4537 to (-20.01, 61.42, -40) mm, rotated rx -180 ry 0 rz 0.01 deg; joints [35.43, -52.281, 121.211, -142.803, 73.574, 168.826]
  MoveL 4538 to (-24, 61.5, -40) mm, rotated rx 180 ry 0 rz 0.01 deg; joints [35.331, -52.161, 120.939, -142.876, 73.432, 168.76]
  MoveL 4539 to (-24.25, 61.5, -40) mm, rotated rx -180 ry 0 rz 0.01 deg; joints [35.325, -52.153, 120.922, -142.881, 73.423, 168.756]
  MoveL 4540 to (-26.43, 61.38, -40) mm, rotated rx 180 ry 0 rz 0.01 deg; joints [35.265, -52.09, 120.781, -142.927, 73.347, 168.725]
  MoveL 4541 to (-26.85, 61.33, -40) mm, rotated rx 180 ry 0 rz 0.01 deg; joints [35.253, -52.079, 120.755, -142.938, 73.333, 168.719]
  MoveL 4542 to (-31.57, 60.47, -40) mm, rotated rx -180 ry 0 rz 0.01 deg; joints [35.103, -51.955, 120.477, -143.062, 73.177, 168.668]
  MoveL 4543 to (-32.21, 60.29, -40) mm, rotated rx -180 ry 0 rz 0.01 deg; joints [35.08, -51.939, 120.442, -143.082, 73.157, 168.663]
  MoveL 4544 to (-34.02, 59.57, -40) mm, rotated rx 180 ry 0 rz 0.01 deg; joints [35.009, -51.899, 120.353, -143.146, 73.102, 168.655]
  MoveL 4545 to (-34.16, 59.51, -40) mm, rotated rx -180 ry 0 rz 0.01 deg; joints [35.003, -51.896, 120.346, -143.151, 73.098, 168.654]
  MoveL 4546 to (-39.24, 57.22, -40) mm, rotated rx -180 ry 0 rz 0.01 deg; joints [34.795, -51.788, 120.109, -143.34, 72.948, 168.637]
  MoveL 4547 to (-39.74, 56.95, -40) mm, rotated rx 180 ry 0 rz 0.01 deg; joints [34.773, -51.779, 120.088, -143.361, 72.934, 168.637]
  MoveL 4548 to (-42.34, 55.21, -40) mm, rotated rx 180 ry 0 rz 0.01 deg; joints [34.646, -51.734, 119.993, -143.481, 72.865, 168.645]
  MoveL 4549 to (-42.66, 54.96, -40) mm, rotated rx 180 ry 0 rz 0.01 deg; joints [34.629, -51.729, 119.982, -143.497, 72.857, 168.647]
  MoveL 4550 to (-44.78, 53.15, -40) mm, rotated rx 180 ry 0 rz 0.01 deg; joints [34.511, -51.701, 119.923, -143.611, 72.806, 168.664]
  MoveL 4551 to (-44.96, 52.98, -40) mm, rotated rx -180 ry 0 rz 0.01 deg; joints [34.501, -51.699, 119.918, -143.621, 72.802, 168.666]
  MoveL 4552 to (-46.05, 51.9, -40) mm, rotated rx 180 ry 0 rz 0.01 deg; joints [34.435, -51.687, 119.894, -143.686, 72.778, 168.679]
  MoveL 4553 to (-46.34, 51.56, -40) mm, rotated rx 180 ry 0 rz 0.01 deg; joints [34.416, -51.685, 119.89, -143.705, 72.772, 168.683]
  MoveL 4554 to (-50.39, 46.33, -40) mm, rotated rx 180 ry 0 rz 0.01 deg; joints [34.128, -51.665, 119.857, -143.997, 72.698, 168.765]
  MoveL 4555 to (-50.64, 45.95, -40) mm, rotated rx 180 ry 0 rz 0.01 deg; joints [34.109, -51.665, 119.857, -144.017, 72.694, 168.772]
  MoveL 4556 to (-68.79, 14.55, -40) mm, rotated rx 180 ry 0 rz 0.01 deg; joints [32.532, -51.709, 120.027, -145.654, 72.461, 169.349]
  MoveL 4557 to (-68.98, 14.18, -40) mm, rotated rx -180 ry 0 rz 0.01 deg; joints [32.514, -51.71, 120.031, -145.673, 72.459, 169.356]
  MoveL 4558 to (-70.67, 10.19, -40) mm, rotated rx -180 ry 0 rz 0.01 deg; joints [32.327, -51.732, 120.089, -145.871, 72.45, 169.437]
  MoveL 4559 to (-70.71, 10.09, -40) mm, rotated rx -180 ry 0 rz 0.01 deg; joints [32.323, -51.733, 120.091, -145.876, 72.45, 169.439]
  MoveL 4560 to (-71.83, 7.18, -40) mm, rotated rx 180 ry 0 rz 0.01 deg; joints [32.189, -51.752, 120.141, -146.018, 72.448, 169.5]
  MoveL 4561 to (-71.98, 6.67, -40) mm, rotated rx 180 ry 0 rz 0.01 deg; joints [32.167, -51.756, 120.153, -146.043, 72.449, 169.511]
  MoveL 4562 to (-72.6, 3.77, -40) mm, rotated rx -180 ry 0 rz 0.01 deg; joints [32.045, -51.791, 120.237, -146.176, 72.466, 169.579]
  MoveL 4563 to (-72.66, 3.38, -40) mm, rotated rx 180 ry 0 rz 0.01 deg; joints [32.03, -51.796, 120.25, -146.194, 72.469, 169.589]
  MoveL 4564 to (-72.94, 0.48, -40) mm, rotated rx 180 ry 0 rz 0.01 deg; joints [31.916, -51.841, 120.357, -146.322, 72.498, 169.662]
  MoveL 4565 to (-72.95, 0.22, -40) mm, rotated rx -180 ry 0 rz 0.01 deg; joints [31.905, -51.845, 120.368, -146.333, 72.501, 169.669]
  MoveL 4566 to (-72.97, -1.24, -40) mm, rotated rx -180 ry 0 rz 0.01 deg; joints [31.851, -51.871, 120.43, -146.395, 72.52, 169.707]
  MoveL 4567 to (-72.95, -1.67, -40) mm, rotated rx 180 ry 0 rz 0.01 deg; joints [31.835, -51.88, 120.45, -146.413, 72.526, 169.719]
  MoveL 4568 to (-72.17, -8.56, -40) mm, rotated rx 180 ry 0 rz 0.01 deg; joints [31.596, -52.03, 120.804, -146.694, 72.649, 169.913]
  MoveL 4569 to (-72, -9.3, -40) mm, rotated rx -180 ry 0 rz 0.01 deg; joints [31.573, -52.048, 120.848, -146.723, 72.665, 169.935]
  MoveL 4570 to (-70.79, -12.75, -40) mm, rotated rx 180 ry 0 rz 0.01 deg; joints [31.471, -52.148, 121.081, -146.849, 72.757, 170.043]
  MoveL 4571 to (-70.74, -12.89, -40) mm, rotated rx -180 ry 0 rz 0.01 deg; joints [31.467, -52.152, 121.091, -146.855, 72.761, 170.048]
  MoveL 4572 to (-69.92, -14.93, -40) mm, rotated rx -180 ry 0 rz 0.01 deg; joints [31.409, -52.215, 121.237, -146.928, 72.82, 170.114]
  MoveL 4573 to (-69.71, -15.35, -40) mm, rotated rx -180 ry 0 rz 0.01 deg; joints [31.398, -52.228, 121.269, -146.943, 72.833, 170.128]
  MoveL 4574 to (-67.66, -18.93, -40) mm, rotated rx 180 ry 0 rz 0.01 deg; joints [31.31, -52.356, 121.567, -147.061, 72.958, 170.252]
  MoveL 4575 to (-67.53, -19.14, -40) mm, rotated rx 180 ry 0 rz 0.01 deg; joints [31.306, -52.364, 121.584, -147.068, 72.966, 170.259]
  MoveL 4576 to (-66.78, -20.25, -40) mm, rotated rx 180 ry 0 rz 0.01 deg; joints [31.281, -52.407, 121.684, -147.103, 73.009, 170.299]
  MoveL 4577 to (-66.29, -20.83, -40) mm, rotated rx -180 ry 0 rz 0.01 deg; joints [31.27, -52.432, 121.743, -147.119, 73.035, 170.322]
  MoveL 4578 to (-59.76, -26.98, -40) mm, rotated rx 180 ry 0 rz 0.01 deg; joints [31.187, -52.742, 122.462, -147.271, 73.362, 170.578]
  MoveL 4579 to (-59.6, -27.12, -40) mm, rotated rx -180 ry 0 rz 0.01 deg; joints [31.185, -52.75, 122.479, -147.275, 73.37, 170.584]
  MoveL 4580 to (-58.51, -28.02, -40) mm, rotated rx 180 ry 0 rz 0.01 deg; joints [31.176, -52.799, 122.593, -147.295, 73.423, 170.624]
  MoveC 4581 to (-58.08, -28.32, -40) mm, rotated rx -180 ry 0 rz 0.01 deg; joints [31.174, -52.818, 122.636, -147.3, 73.444, 170.638] to (-57.61, -28.56, -40) mm, rotated rx -180 ry 0 rz 0.01 deg; joints [31.176, -52.836, 122.679, -147.302, 73.464, 170.651]
  MoveL 4582 to (-50.81, -31.27, -40) mm, rotated rx 180 ry 0 rz 0.01 deg; joints [31.23, -53.092, 123.268, -147.3, 73.755, 170.823]
  MoveL 4583 to (-342.73, -31.27, -40) mm, rotated rx -180 ry 0 rz 0.01 deg; joints [25.561, -42.842, 100.722, -150.713, 61.939, 166.303]
  MoveL 4584 to (-336.29, -28.75, -40) mm, rotated rx 180 ry 0 rz 0.01 deg; joints [25.75, -43.054, 101.172, -150.568, 62.196, 166.337]
  MoveL 4585 to (-335.79, -28.51, -40) mm, rotated rx 180 ry 0 rz 0.01 deg; joints [25.767, -43.07, 101.205, -150.554, 62.215, 166.338]
  MoveL 4586 to (-335.06, -28.08, -40) mm, rotated rx 180 ry 0 rz 0.01 deg; joints [25.793, -43.091, 101.25, -150.532, 62.242, 166.337]
  MoveL 4587 to (-334.48, -27.64, -40) mm, rotated rx -180 ry 0 rz 0.01 deg; joints [25.817, -43.106, 101.281, -150.509, 62.263, 166.333]
  MoveL 4588 to (-327.58, -21.19, -40) mm, rotated rx -180 ry 0 rz 0.01 deg; joints [26.149, -43.262, 101.603, -150.191, 62.493, 166.255]
  MoveL 4589 to (-327.36, -20.97, -40) mm, rotated rx 180 ry 0 rz 0.01 deg; joints [26.16, -43.266, 101.612, -150.18, 62.501, 166.252]
  MoveL 4590 to (-326.73, -20.25, -40) mm, rotated rx 180 ry 0 rz 0.01 deg; joints [26.195, -43.278, 101.636, -150.146, 62.52, 166.241]
  MoveL 4591 to (-326.35, -19.74, -40) mm, rotated rx 180 ry 0 rz 0.01 deg; joints [26.218, -43.284, 101.647, -150.121, 62.531, 166.232]
  MoveL 4592 to (-324.17, -16.08, -40) mm, rotated rx -180 ry 0 rz 0.01 deg; joints [26.378, -43.302, 101.679, -149.951, 62.585, 166.158]
  MoveL 4593 to (-324.03, -15.82, -40) mm, rotated rx 180 ry 0 rz 0.01 deg; joints [26.389, -43.303, 101.68, -149.939, 62.588, 166.152]
  MoveL 4594 to (-323.37, -14.46, -40) mm, rotated rx 180 ry 0 rz 0.01 deg; joints [26.446, -43.303, 101.678, -149.877, 62.601, 166.122]
  MoveL 4595 to (-323.24, -14.13, -40) mm, rotated rx 180 ry 0 rz 0.01 deg; joints [26.46, -43.302, 101.676, -149.862, 62.603, 166.114]
  MoveL 4596 to (-321.51, -9.32, -40) mm, rotated rx -180 ry 0 rz 0.01 deg; joints [26.65, -43.28, 101.619, -149.645, 62.623, 165.997]
  MoveL 4597 to (-321.34, -8.59, -40) mm, rotated rx 180 ry 0 rz 0.01 deg; joints [26.678, -43.273, 101.602, -149.613, 62.623, 165.978]
  MoveL 4598 to (-320.68, -3.15, -40) mm, rotated rx -180 ry 0 rz 0.01 deg; joints [26.872, -43.196, 101.426, -149.377, 62.589, 165.822]
  MoveL 4599 to (-320.67, -2.97, -40) mm, rotated rx -180 ry 0 rz 0.01 deg; joints [26.878, -43.193, 101.42, -149.369, 62.587, 165.817]
  MoveL 4600 to (-320.52, -0.8, -40) mm, rotated rx -180 ry 0 rz 0.01 deg; joints [26.953, -43.157, 101.339, -149.275, 62.569, 165.752]
  MoveL 4601 to (-320.52, -0.31, -40) mm, rotated rx 180 ry 0 rz 0.01 deg; joints [26.97, -43.148, 101.318, -149.254, 62.563, 165.737]
  MoveL 4602 to (-320.74, 2.59, -40) mm, rotated rx 180 ry 0 rz 0.01 deg; joints [27.063, -43.083, 101.174, -149.132, 62.52, 165.644]
  MoveL 4603 to (-320.79, 2.98, -40) mm, rotated rx -180 ry 0 rz 0.01 deg; joints [27.075, -43.074, 101.153, -149.116, 62.514, 165.631]
  MoveL 4604 to (-321.35, 5.88, -40) mm, rotated rx 180 ry 0 rz 0.01 deg; joints [27.162, -42.996, 100.98, -148.996, 62.456, 165.531]
  MoveL 4605 to (-321.42, 6.16, -40) mm, rotated rx 180 ry 0 rz 0.01 deg; joints [27.17, -42.988, 100.962, -148.984, 62.45, 165.521]
  MoveL 4606 to (-321.82, 7.58, -40) mm, rotated rx -180 ry 0 rz 0.01 deg; joints [27.211, -42.944, 100.865, -148.926, 62.416, 165.47]
  MoveL 4607 to (-321.95, 7.95, -40) mm, rotated rx -180 ry 0 rz 0.01 deg; joints [27.221, -42.932, 100.839, -148.912, 62.406, 165.456]
  MoveL 4608 to (-324.35, 13.78, -40) mm, rotated rx -180 ry 0 rz 0.01 deg; joints [27.373, -42.722, 100.379, -148.678, 62.234, 165.231]
  MoveL 4609 to (-324.54, 14.18, -40) mm, rotated rx 180 ry 0 rz 0.01 deg; joints [27.383, -42.707, 100.344, -148.662, 62.221, 165.215]
  MoveL 4610 to (-342.68, 45.66, -40) mm, rotated rx 180 ry 0 rz 0.01 deg; joints [28.1, -41.337, 97.361, -147.421, 61.06, 163.867]
  MoveL 4611 to (-342.91, 46, -40) mm, rotated rx 180 ry 0 rz 0.01 deg; joints [28.107, -41.321, 97.326, -147.408, 61.046, 163.851]
  MoveL 4612 to (-344.86, 48.62, -40) mm, rotated rx -180 ry 0 rz 0.01 deg; joints [28.158, -41.186, 97.034, -147.306, 60.929, 163.727]
  MoveL 4613 to (-344.92, 48.69, -40) mm, rotated rx -180 ry 0 rz 0.01 deg; joints [28.159, -41.182, 97.026, -147.303, 60.925, 163.724]
  MoveL 4614 to (-347.45, 51.89, -40) mm, rotated rx -180 ry 0 rz 0.01 deg; joints [28.219, -41.011, 96.656, -147.178, 60.776, 163.568]
  MoveL 4615 to (-347.83, 52.3, -40) mm, rotated rx -180 ry 0 rz 0.01 deg; joints [28.225, -40.987, 96.604, -147.163, 60.755, 163.547]
  MoveL 4616 to (-350.27, 54.51, -40) mm, rotated rx 180 ry 0 rz 0.01 deg; joints [28.254, -40.839, 96.286, -147.079, 60.621, 163.426]
  MoveL 4617 to (-350.6, 54.78, -40) mm, rotated rx 180 ry 0 rz 0.01 deg; joints [28.257, -40.82, 96.244, -147.069, 60.603, 163.41]
  MoveL 4618 to (-352.99, 56.46, -40) mm, rotated rx 180 ry 0 rz 0.01 deg; joints [28.269, -40.685, 95.955, -147.008, 60.477, 163.307]
  MoveL 4619 to (-353.26, 56.62, -40) mm, rotated rx -180 ry 0 rz 0.01 deg; joints [28.27, -40.671, 95.924, -147.002, 60.463, 163.296]
  MoveL 4620 to (-354.71, 57.45, -40) mm, rotated rx -180 ry 0 rz 0.01 deg; joints [28.272, -40.593, 95.757, -146.973, 60.389, 163.239]
  MoveL 4621 to (-355.03, 57.61, -40) mm, rotated rx 180 ry 0 rz 0.01 deg; joints [28.271, -40.576, 95.721, -146.968, 60.373, 163.228]
  MoveL 4622 to (-360.84, 60.14, -40) mm, rotated rx 180 ry 0 rz 0.01 deg; joints [28.252, -40.28, 95.088, -146.883, 60.085, 163.026]
  MoveL 4623 to (-361.55, 60.36, -40) mm, rotated rx -180 ry 0 rz 0.01 deg; joints [28.247, -40.245, 95.015, -146.876, 60.05, 163.004]
  MoveL 4624 to (-365.9, 61.2, -40) mm, rotated rx 180 ry 0 rz 0.01 deg; joints [28.2, -40.045, 94.587, -146.857, 59.846, 162.888]
  MoveL 4625 to (-366.16, 61.24, -40) mm, rotated rx 180 ry 0 rz 0.01 deg; joints [28.197, -40.033, 94.562, -146.856, 59.833, 162.881]
  MoveL 4626 to (-368.34, 61.49, -40) mm, rotated rx -180 ry 0 rz 0.01 deg; joints [28.167, -39.936, 94.356, -146.853, 59.733, 162.828]
  MoveL 4627 to (-368.78, 61.51, -40) mm, rotated rx -180 ry 0 rz 0.01 deg; joints [28.161, -39.917, 94.316, -146.854, 59.713, 162.819]
  MoveL 4628 to (-373.5, 61.42, -40) mm, rotated rx -180 ry 0 rz 0.01 deg; joints [28.078, -39.719, 93.897, -146.873, 59.501, 162.725]
  MoveL 4629 to (-374.4, 61.28, -40) mm, rotated rx 180 ry 0 rz 0.01 deg; joints [28.059, -39.684, 93.823, -146.882, 59.462, 162.712]
  MoveL 4630 to (-383.59, 58.54, -40) mm, rotated rx -180 ry 0 rz 0.01 deg; joints [27.819, -39.351, 93.123, -147.028, 59.078, 162.617]
  MoveL 4631 to (-383.92, 58.42, -40) mm, rotated rx 180 ry 0 rz 0.01 deg; joints [27.809, -39.34, 93.099, -147.034, 59.064, 162.614]
  MoveL 4632 to (-384.92, 58.01, -40) mm, rotated rx 180 ry 0 rz 0.01 deg; joints [27.78, -39.306, 93.028, -147.054, 59.023, 162.608]
  MoveL 4633 to (-385.72, 57.54, -40) mm, rotated rx -180 ry 0 rz 0.01 deg; joints [27.752, -39.282, 92.978, -147.077, 58.992, 162.607]
  MoveL 4634 to (-393.65, 51.26, -40) mm, rotated rx 180 ry 0 rz 0.01 deg; joints [27.423, -39.076, 92.553, -147.369, 58.703, 162.66]
  MoveL 4635 to (-394.11, 50.81, -40) mm, rotated rx -180 ry 0 rz 0.01 deg; joints [27.402, -39.065, 92.531, -147.389, 58.687, 162.666]
  MoveL 4636 to (-395.22, 49.53, -40) mm, rotated rx 180 ry 0 rz 0.01 deg; joints [27.343, -39.045, 92.491, -147.447, 58.651, 162.688]
  MoveL 4637 to (-395.51, 49.14, -40) mm, rotated rx -180 ry 0 rz 0.01 deg; joints [27.326, -39.041, 92.483, -147.465, 58.642, 162.695]
  MoveL 4638 to (-397.82, 45.51, -40) mm, rotated rx 180 ry 0 rz 0.01 deg; joints [27.174, -39.018, 92.442, -147.627, 58.578, 162.773]
  MoveL 4639 to (-397.89, 45.4, -40) mm, rotated rx -180 ry 0 rz 0.01 deg; joints [27.17, -39.018, 92.441, -147.632, 58.576, 162.776]
  MoveL 4640 to (-401.77, 38.76, -40) mm, rotated rx 180 ry 0 rz 0.01 deg; joints [26.897, -38.991, 92.395, -147.929, 58.474, 162.925]
  MoveL 4641 to (-402, 38.3, -40) mm, rotated rx 180 ry 0 rz 0.01 deg; joints [26.879, -38.991, 92.396, -147.949, 58.469, 162.936]
  MoveL 4642 to (-402.54, 36.92, -40) mm, rotated rx -180 ry 0 rz 0.01 deg; joints [26.827, -38.996, 92.409, -148.01, 58.459, 162.972]
  MoveL 4643 to (-402.69, 36.46, -40) mm, rotated rx 180 ry 0 rz 0.01 deg; joints [26.81, -38.999, 92.417, -148.031, 58.458, 162.985]
  MoveL 4644 to (-403.78, 31.9, -40) mm, rotated rx -180 ry 0 rz 0.01 deg; joints [26.648, -39.048, 92.528, -148.231, 58.46, 163.12]
  MoveL 4645 to (-403.79, 333.8, -40) mm, rotated rx -180 ry 0 rz 0.01 deg; joints [35.412, -30.81, 74.811, -134.71, 54.648, 150.634]
  MoveL 4646 to (-403.73, 334.87, -40) mm, rotated rx 180 ry 0 rz 0.01 deg; joints [35.442, -30.776, 74.738, -134.66, 54.636, 150.582]
  MoveL 4647 to (-403.53, 335.74, -40) mm, rotated rx 180 ry 0 rz 0.01 deg; joints [35.468, -30.755, 74.695, -134.62, 54.633, 150.546]
  MoveL 4648 to (-403.42, 336, -40) mm, rotated rx -180 ry 0 rz 0.01 deg; joints [35.477, -30.752, 74.687, -134.608, 54.635, 150.536]
  MoveL 4649 to (-403.03, 336.5, -39.83) mm, rotated rx 180 ry 0 rz 0.01 deg; joints [35.498, -30.761, 74.691, -134.585, 54.642, 150.519]
  MoveL 4650 to (-402.62, 336.71, -39.37) mm, rotated rx -180 ry 0 rz 0.01 deg; joints [35.511, -30.794, 74.72, -134.569, 54.646, 150.508]
  MoveL 4651 to (-402.46, 336.75, -38.73) mm, rotated rx -180 ry 0 rz 0.01 deg; joints [35.515, -30.828, 74.738, -134.557, 54.636, 150.491]
  Set speed (1000.0 mm/s)
  MoveL 4652 to (-402.46, 336.75, 11) mm, rotated rx 180 ry 0 rz 0.01 deg; joints [35.493, -32.912, 74.899, -133.574, 53.288, 148.796]
  Set speed (1000.0 mm/s)
  MoveL 4653 to (-176.91, 111.47, 11) mm, rotated rx 180 ry 0 rz 0.01 deg; joints [33.429, -48.887, 107.782, -142.569, 65.053, 163.079]
  Set speed (1000.0 mm/s)
  MoveL 4654 to (-176.91, 111.47, -28.23) mm, rotated rx 180 ry 0 rz 0.01 deg; joints [33.451, -46.81, 107.683, -143.082, 66.636, 164.379]
  Set speed (100.0 mm/s)
  MoveL 4655 to (-176.83, 111.56, -28.78) mm, rotated rx 180 ry 0 rz 0.01 deg; joints [33.456, -46.781, 107.682, -143.084, 66.659, 164.395]
  MoveL 4656 to (-176.61, 111.83, -29.22) mm, rotated rx -180 ry 0 rz 0.01 deg; joints [33.47, -46.759, 107.683, -143.076, 66.682, 164.404]
  MoveL 4657 to (-176.4, 112.12, -29.42) mm, rotated rx 180 ry 0 rz 0.01 deg; joints [33.484, -46.749, 107.683, -143.064, 66.694, 164.405]
  MoveL 4658 to (-176.2, 112.46, -29.5) mm, rotated rx 180 ry 0 rz 0.01 deg; joints [33.5, -46.744, 107.682, -143.048, 66.701, 164.4]
  MoveL 4659 to (-176.62, 119.1, -29.75) mm, rotated rx 180 ry 0 rz 0.01 deg; joints [33.708, -46.567, 107.316, -142.783, 66.612, 164.189]
  MoveL 4660 to (-182.9, 121.31, -29.99) mm, rotated rx 180 ry 0 rz 0.01 deg; joints [33.644, -46.282, 106.73, -142.77, 66.353, 164.017]
  MoveL 4661 to (-187.39, 116.41, -30.24) mm, rotated rx 180 ry 0 rz 0.01 deg; joints [33.388, -46.22, 106.633, -143.028, 66.249, 164.105]
  MoveL 4662 to (-184.65, 110.35, -30.48) mm, rotated rx -180 ry 0 rz 0.01 deg; joints [33.249, -46.44, 107.143, -143.249, 66.44, 164.354]
  MoveL 4663 to (-178, 110.49, -30.73) mm, rotated rx -180 ry 0 rz 0.01 deg; joints [33.397, -46.659, 107.638, -143.166, 66.705, 164.472]
  MoveL 4664 to (-175.52, 116.66, -30.98) mm, rotated rx 180 ry 0 rz 0.01 deg; joints [33.653, -46.594, 107.516, -142.885, 66.733, 164.326]
  MoveL 4665 to (-180.22, 121.36, -31.22) mm, rotated rx 180 ry 0 rz 0.01 deg; joints [33.704, -46.31, 106.924, -142.751, 66.503, 164.101]
  MoveL 4666 to (-186.39, 118.89, -31.47) mm, rotated rx 180 ry 0 rz 0.01 deg; joints [33.491, -46.134, 106.579, -142.929, 66.305, 164.081]
  MoveL 4667 to (-186.54, 112.24, -31.71) mm, rotated rx 180 ry 0 rz 0.01 deg; joints [33.271, -46.265, 106.9, -143.208, 66.392, 164.3]
  MoveL 4668 to (-180.48, 109.5, -31.96) mm, rotated rx 180 ry 0 rz 0.01 deg; joints [33.311, -46.527, 107.494, -143.252, 66.67, 164.5]
  MoveL 4669 to (-175.58, 113.99, -32.2) mm, rotated rx -180 ry 0 rz 0.01 deg; joints [33.565, -46.586, 107.64, -143.011, 66.813, 164.449]
  MoveL 4670 to (-177.79, 120.26, -32.45) mm, rotated rx -180 ry 0 rz 0.01 deg; joints [33.722, -46.355, 107.158, -142.782, 66.659, 164.219]
  MoveL 4671 to (-184.42, 120.69, -32.7) mm, rotated rx -180 ry 0 rz 0.01 deg; joints [33.592, -46.098, 106.633, -142.847, 66.407, 164.097]
  MoveL 4672 to (-187.43, 114.76, -32.94) mm, rotated rx 180 ry 0 rz 0.01 deg; joints [33.335, -46.112, 106.701, -143.13, 66.374, 164.243]
  MoveL 4673 to (-183.15, 109.67, -33.19) mm, rotated rx -180 ry 0 rz 0.01 deg; joints [33.26, -46.363, 107.278, -143.292, 66.613, 164.487]
  MoveL 4674 to (-176.79, 111.61, -33.43) mm, rotated rx 180 ry 0 rz 0.01 deg; joints [33.461, -46.531, 107.662, -143.139, 66.845, 164.544]
  MoveL 4675 to (-176.07, 118.22, -33.68) mm, rotated rx -180 ry 0 rz 0.01 deg; joints [33.693, -46.395, 107.385, -142.861, 66.799, 164.353]
  MoveL 4676 to (-181.87, 121.47, -33.93) mm, rotated rx 180 ry 0 rz 0.01 deg; joints [33.674, -46.105, 106.782, -142.8, 66.544, 164.156]
  MoveL 4677 to (-187.14, 117.42, -34.17) mm, rotated rx -180 ry 0 rz 0.01 deg; joints [33.428, -45.997, 106.584, -143.032, 66.4, 164.202]
  MoveL 4678 to (-185.48, 110.98, -34.42) mm, rotated rx 180 ry 0 rz 0.01 deg; joints [33.254, -46.186, 107.031, -143.281, 66.555, 164.444]
  MoveL 4679 to (-178.91, 109.98, -34.66) mm, rotated rx 180 ry 0 rz 0.01 deg; joints [33.363, -46.427, 107.578, -143.246, 66.832, 164.598]
  MoveL 4680 to (-175.4, 115.63, -34.91) mm, rotated rx 180 ry 0 rz 0.01 deg; joints [33.624, -46.41, 107.559, -142.974, 66.906, 164.487]
  MoveL 4681 to (-179.22, 121.07, -35.16) mm, rotated rx -180 ry 0 rz 0.01 deg; joints [33.718, -46.141, 106.996, -142.8, 66.7, 164.254]
  MoveL 4682 to (-185.73, 119.69, -35.4) mm, rotated rx -180 ry 0 rz 0.01 deg; joints [33.533, -45.93, 106.571, -142.937, 66.475, 164.192]
  MoveL 4683 to (-187.02, 113.17, -35.65) mm, rotated rx -180 ry 0 rz 0.01 deg; joints [33.293, -46.017, 106.799, -143.223, 66.516, 164.387]
  MoveL 4684 to (-181.52, 109.42, -35.89) mm, rotated rx 180 ry 0 rz 0.01 deg; joints [33.289, -46.281, 107.401, -143.315, 66.786, 164.609]
  MoveL 4685 to (-175.92, 113.01, -36.14) mm, rotated rx -180 ry 0 rz 0.01 deg; joints [33.527, -46.384, 107.645, -143.103, 66.968, 164.6]
  MoveL 4686 to (-177.02, 119.56, -36.39) mm, rotated rx 180 ry 0 rz 0.01 deg; joints [33.718, -46.186, 107.233, -142.85, 66.852, 164.38]
  MoveL 4687 to (-183.48, 121.13, -36.63) mm, rotated rx 180 ry 0 rz 0.01 deg; joints [33.629, -45.911, 106.664, -142.866, 66.592, 164.225]
  MoveL 4688 to (-187.46, 115.8, -36.88) mm, rotated rx -180 ry 0 rz 0.01 deg; joints [33.37, -45.877, 106.628, -143.135, 66.514, 164.334]
  MoveL 4689 to (-184.12, 110.05, -37.12) mm, rotated rx 180 ry 0 rz 0.01 deg; joints [33.254, -46.11, 107.167, -143.335, 66.726, 164.583]
  MoveL 4690 to (-177.52, 110.86, -37.37) mm, rotated rx -180 ry 0 rz 0.01 deg; joints [33.423, -46.31, 107.625, -143.225, 66.982, 164.68]
  MoveL 4691 to (-175.68, 117.25, -37.61) mm, rotated rx -180 ry 0 rz 0.01 deg; joints [33.673, -46.219, 107.444, -142.943, 66.981, 164.517]
  MoveL 4692 to (-180.83, 121.46, -37.86) mm, rotated rx -180 ry 0 rz 0.01 deg; joints [33.698, -45.931, 106.843, -142.836, 66.738, 164.3]
  MoveL 4693 to (-186.71, 118.37, -38.11) mm, rotated rx -180 ry 0 rz 0.01 deg; joints [33.47, -45.78, 106.55, -143.035, 66.558, 164.303]
  MoveL 4694 to (-186.19, 111.74, -38.35) mm, rotated rx 180 ry 0 rz 0.01 deg; joints [33.266, -45.933, 106.92, -143.305, 66.673, 164.532]
  MoveL 4695 to (-179.89, 109.62, -38.6) mm, rotated rx 180 ry 0 rz 0.01 deg; joints [33.332, -46.188, 107.502, -143.32, 66.954, 164.717]
  MoveL 4696 to (-175.46, 114.59, -38.84) mm, rotated rx 180 ry 0 rz 0.01 deg; joints [33.591, -46.219, 107.587, -143.064, 67.072, 164.644]
  MoveL 4697 to (-178.29, 120.6, -39.09) mm, rotated rx 180 ry 0 rz 0.01 deg; joints [33.726, -45.973, 107.071, -142.855, 66.895, 164.411]
  MoveL 4698 to (-184.94, 120.37, -39.34) mm, rotated rx 180 ry 0 rz 0.01 deg; joints [33.574, -45.732, 106.579, -142.947, 66.65, 164.309]
  MoveL 4699 to (-187.33, 114.16, -39.58) mm, rotated rx 180 ry 0 rz 0.01 deg; joints [33.321, -45.774, 106.707, -143.233, 66.646, 164.473]
  MoveL 4700 to (-182.56, 109.53, -39.83) mm, rotated rx 180 ry 0 rz 0.01 deg; joints [33.272, -46.03, 107.298, -143.37, 66.9, 164.712]
  MoveL 4701 to (-176.42, 112.09, -40.07) mm, rotated rx -180 ry 0 rz 0.01 deg; joints [33.489, -46.174, 107.633, -143.193, 67.115, 164.745]
  MoveL 4702 to (-176.38, 118.74, -40.32) mm, rotated rx 180 ry 0 rz 0.01 deg; joints [33.707, -46.015, 107.303, -142.923, 67.041, 164.543]
  MoveL 4703 to (-182.47, 121.4, -40.57) mm, rotated rx -180 ry 0 rz 0.01 deg; joints [33.662, -45.73, 106.707, -142.89, 66.781, 164.359]
  MoveL 4704 to (-187.31, 116.83, -40.81) mm, rotated rx 180 ry 0 rz 0.01 deg; joints [33.409, -45.649, 106.568, -143.138, 66.66, 164.427]
  MoveL 4705 to (-185.01, 110.59, -41.06) mm, rotated rx 180 ry 0 rz 0.01 deg; joints [33.255, -45.855, 107.053, -143.37, 66.839, 164.674]
  MoveL 4706 to (-178.37, 110.26, -41.3) mm, rotated rx -180 ry 0 rz 0.01 deg; joints [33.387, -46.081, 107.571, -143.307, 67.112, 164.808]
  MoveL 4707 to (-175.45, 116.23, -41.55) mm, rotated rx 180 ry 0 rz 0.01 deg; joints [33.646, -46.037, 107.492, -143.029, 67.157, 164.678]
  MoveL 4708 to (-179.8, 121.26, -41.8) mm, rotated rx 180 ry 0 rz 0.01 deg; joints [33.716, -45.76, 106.91, -142.878, 66.934, 164.449]
  MoveL 4709 to (-186.13, 119.24, -42.04) mm, rotated rx 180 ry 0 rz 0.01 deg; joints [33.513, -45.571, 106.53, -143.04, 66.723, 164.41]
  MoveL 4710 to (-186.76, 112.62, -42.29) mm, rotated rx 180 ry 0 rz 0.01 deg; joints [33.284, -45.683, 106.813, -143.323, 66.793, 164.617]
  MoveL 4711 to (-180.91, 109.44, -42.53) mm, rotated rx -180 ry 0 rz 0.01 deg; joints [33.306, -45.944, 107.413, -143.386, 67.071, 164.828]
  MoveL 4712 to (-175.7, 113.57, -42.78) mm, rotated rx 180 ry 0 rz 0.01 deg; joints [33.555, -46.02, 107.6, -143.155, 67.23, 164.797]
  MoveL 4713 to (-177.45, 119.99, -43.02) mm, rotated rx -180 ry 0 rz 0.01 deg; joints [33.726, -45.804, 107.145, -142.917, 67.089, 164.57]
  MoveL 4714 to (-184.04, 120.89, -43.27) mm, rotated rx 180 ry 0 rz 0.01 deg; joints [33.613, -45.541, 106.6, -142.962, 66.831, 164.432]
  MoveL 4715 to (-187.46, 115.19, -43.52) mm, rotated rx 180 ry 0 rz 0.01 deg; joints [33.354, -45.535, 106.624, -143.239, 66.78, 164.561]
  MoveL 4716 to (-183.56, 109.81, -43.76) mm, rotated rx 180 ry 0 rz 0.01 deg; joints [33.262, -45.777, 107.188, -143.417, 67.012, 164.809]
  MoveL 4717 to (-177.08, 111.28, -44.01) mm, rotated rx -180 ry 0 rz 0.01 deg; joints [33.45, -45.957, 107.604, -143.281, 67.255, 164.884]
  MoveL 4718 to (-175.89, 117.82, -44.25) mm, rotated rx 180 ry 0 rz 0.01 deg; joints [33.69, -45.84, 107.365, -143.001, 67.226, 164.705]
  MoveL 4719 to (-181.43, 121.49, -44.5) mm, rotated rx -180 ry 0 rz 0.01 deg; joints [33.689, -45.553, 106.761, -142.921, 66.972, 164.498]
  MoveL 4720 to (-214.17, 121.49, -44.5) mm, rotated rx -180 ry 0 rz 0.01 deg; joints [32.993, -44.393, 104.247, -143.291, 65.683, 163.909]
  MoveC 4721 to (-216.09, 120.38, -44.5) mm, rotated rx 180 ry 0 rz 0.01 deg; joints [32.917, -44.349, 104.153, -143.357, 65.621, 163.91] to (-216.09, 118.16, -44.5) mm, rotated rx 180 ry 0 rz 0.01 deg; joints [32.846, -44.399, 104.264, -143.448, 65.649, 163.983]
  MoveL 4722 to (-214.87, 116.03, -44.5) mm, rotated rx -180 ry 0 rz 0.01 deg; joints [32.803, -44.49, 104.467, -143.523, 65.725, 164.074]
  MoveC 4723 to (-213.83, 114.99, -44.5) mm, rotated rx -180 ry 0 rz 0.01 deg; joints [32.791, -44.551, 104.6, -143.555, 65.78, 164.126] to (-212.41, 114.61, -44.5) mm, rotated rx 180 ry 0 rz 0.01 deg; joints [32.808, -44.61, 104.729, -143.555, 65.841, 164.164]
  MoveL 4724 to (-181.09, 114.61, -44.5) mm, rotated rx 180 ry 0 rz 0.01 deg; joints [33.473, -45.717, 107.132, -143.199, 67.075, 164.723]
  MoveC 4725 to (-179.67, 114.99, -44.5) mm, rotated rx 180 ry 0 rz 0.01 deg; joints [33.516, -45.758, 107.22, -143.166, 67.125, 164.736] to (-178.63, 116.03, -44.5) mm, rotated rx -180 ry 0 rz 0.01 deg; joints [33.572, -45.771, 107.247, -143.111, 67.152, 164.722]
  MoveL 4726 to (-177.4, 118.15, -44.5) mm, rotated rx 180 ry 0 rz 0.01 deg; joints [33.668, -45.767, 107.233, -143.009, 67.172, 164.676]
  MoveC 4727 to (-177.4, 120.38, -44.5) mm, rotated rx -180 ry 0 rz 0.01 deg; joints [33.741, -45.718, 107.121, -142.918, 67.143, 164.605] to (-179.33, 121.49, -44.5) mm, rotated rx 180 ry 0 rz 0.01 deg; joints [33.735, -45.626, 106.92, -142.896, 67.054, 164.536]
  MoveL 4728 to (-181.43, 121.49, -44.5) mm, rotated rx -180 ry 0 rz 0.01 deg; joints [33.689, -45.553, 106.761, -142.921, 66.972, 164.498]
  MoveC 4729 to (-184.8, 122.51, -44.5) mm, rotated rx -180 ry 0 rz 0.01 deg; joints [33.65, -45.412, 106.454, -142.92, 66.828, 164.406] to (-187.04, 125.22, -44.5) mm, rotated rx 180 ry 0 rz 0.01 deg; joints [33.689, -45.273, 106.146, -142.835, 66.705, 164.279]
  MoveC 4730 to (-189.28, 127.94, -44.5) mm, rotated rx 180 ry 0 rz 0.01 deg; joints [33.729, -45.134, 105.838, -142.749, 66.583, 164.151] to (-192.64, 128.96, -44.5) mm, rotated rx 180 ry 0 rz 0.01 deg; joints [33.689, -44.992, 105.529, -142.747, 66.438, 164.057]
  MoveL 4731 to (-214.9, 128.96, -44.5) mm, rotated rx 180 ry 0 rz 0.01 deg; joints [33.218, -44.198, 103.811, -142.991, 65.559, 163.652]
  MoveC 4732 to (-218.63, 129.07, -44.5) mm, rotated rx -180 ry 0 rz 0.01 deg; joints [33.143, -44.061, 103.514, -143.025, 65.409, 163.579] to (-222.35, 129.39, -44.5) mm, rotated rx -180 ry 0 rz 0.01 deg; joints [33.076, -43.919, 103.206, -143.049, 65.256, 163.5]
  MoveC 4733 to (-226.06, 129.81, -44.5) mm, rotated rx 180 ry 0 rz 0.01 deg; joints [33.012, -43.774, 102.894, -143.069, 65.102, 163.417] to (-229.77, 130.21, -44.5) mm, rotated rx 180 ry 0 rz 0.01 deg; joints [32.949, -43.629, 102.58, -143.089, 64.948, 163.335]
  MoveC 4734 to (-231.56, 129.29, -44.5) mm, rotated rx -180 ry 0 rz 0.01 deg; joints [32.882, -43.584, 102.485, -143.144, 64.887, 163.331] to (-231.46, 127.28, -44.5) mm, rotated rx -180 ry 0 rz 0.01 deg; joints [32.821, -43.634, 102.596, -143.226, 64.917, 163.4]
  MoveC 4735 to (-228.68, 123.31, -44.5) mm, rotated rx -180 ry 0 rz 0.01 deg; joints [32.751, -43.826, 103.018, -143.363, 65.079, 163.583] to (-226.05, 119.24, -44.5) mm, rotated rx -180 ry 0 rz 0.01 deg; joints [32.675, -44.013, 103.43, -143.505, 65.237, 163.765]
  MoveC 4736 to (-223.54, 115.1, -44.5) mm, rotated rx -180 ry 0 rz 0.01 deg; joints [32.593, -44.198, 103.836, -143.651, 65.39, 163.946] to (-221.09, 110.92, -44.5) mm, rotated rx -180 ry 0 rz 0.01 deg; joints [32.509, -44.38, 104.236, -143.799, 65.542, 164.126]
  MoveC 4737 to (-217.98, 107.81, -44.5) mm, rotated rx 180 ry 0 rz 0.01 deg; joints [32.473, -44.56, 104.634, -143.895, 65.706, 164.283] to (-213.74, 106.67, -44.5) mm, rotated rx -180 ry 0 rz 0.01 deg; joints [32.523, -44.738, 105.021, -143.897, 65.89, 164.396]
  MoveL 4738 to (-179.78, 106.67, -44.5) mm, rotated rx -180 ry 0 rz 0.01 deg; joints [33.241, -45.937, 107.626, -143.509, 67.229, 164.997]
  MoveC 4739 to (-175.53, 107.81, -44.5) mm, rotated rx -180 ry 0 rz 0.01 deg; joints [33.37, -46.06, 107.89, -143.41, 67.38, 165.035] to (-172.41, 110.92, -44.5) mm, rotated rx -180 ry 0 rz 0.01 deg; joints [33.54, -46.099, 107.97, -143.243, 67.46, 164.992]
  MoveC 4740 to (-169.97, 115.09, -44.5) mm, rotated rx 180 ry 0 rz 0.01 deg; joints [33.73, -46.091, 107.946, -143.042, 67.5, 164.903] to (-167.46, 119.23, -44.5) mm, rotated rx -180 ry 0 rz 0.01 deg; joints [33.921, -46.086, 107.926, -142.841, 67.543, 164.816]
  MoveC 4741 to (-164.85, 123.3, -44.5) mm, rotated rx 180 ry 0 rz 0.01 deg; joints [34.111, -46.085, 107.916, -142.641, 67.59, 164.733] to (-162.09, 127.27, -44.5) mm, rotated rx -180 ry 0 rz 0.01 deg; joints [34.302, -46.091, 107.921, -142.443, 67.645, 164.656]
  MoveC 4742 to (-161.98, 129.29, -44.5) mm, rotated rx -180 ry 0 rz 0.01 deg; joints [34.37, -46.049, 107.827, -142.36, 67.622, 164.593] to (-163.78, 130.21, -44.5) mm, rotated rx 180 ry 0 rz 0.01 deg; joints [34.359, -45.967, 107.646, -142.346, 67.541, 164.532]
  MoveC 4743 to (-167.48, 129.81, -44.5) mm, rotated rx 180 ry 0 rz 0.01 deg; joints [34.264, -45.849, 107.39, -142.409, 67.404, 164.48] to (-171.18, 129.39, -44.5) mm, rotated rx 180 ry 0 rz 0.01 deg; joints [34.169, -45.731, 107.134, -142.472, 67.267, 164.427]
  MoveC 4744 to (-174.89, 129.07, -44.5) mm, rotated rx 180 ry 0 rz 0.01 deg; joints [34.077, -45.61, 106.871, -142.531, 67.128, 164.372] to (-178.62, 128.96, -44.5) mm, rotated rx -180 ry 0 rz 0.01 deg; joints [33.993, -45.483, 106.595, -142.581, 66.985, 164.309]
  MoveL 4745 to (-192.64, 128.96, -44.5) mm, rotated rx -180 ry 0 rz 0.01 deg; joints [33.689, -44.992, 105.529, -142.747, 66.438, 164.057]
  MoveC 4746 to (-195.97, 129.96, -44.5) mm, rotated rx -180 ry 0 rz 0.01 deg; joints [33.65, -44.852, 105.223, -142.744, 66.294, 163.965] to (-198.21, 132.62, -44.5) mm, rotated rx 180 ry 0 rz 0.01 deg; joints [33.688, -44.712, 104.916, -142.66, 66.172, 163.837]
  MoveC 4747 to (-200.43, 135.29, -44.5) mm, rotated rx 180 ry 0 rz 0.01 deg; joints [33.726, -44.572, 104.608, -142.575, 66.05, 163.709] to (-203.77, 136.28, -44.5) mm, rotated rx 180 ry 0 rz 0.01 deg; joints [33.686, -44.43, 104.3, -142.571, 65.906, 163.616]
  MoveL 4748 to (-214.9, 136.25, -44.5) mm, rotated rx -180 ry 0 rz 0.01 deg; joints [33.45, -44.032, 103.438, -142.691, 65.466, 163.411]
  MoveC 4749 to (-223.05, 136.54, -44.5) mm, rotated rx -180 ry 0 rz 0.01 deg; joints [33.289, -43.729, 102.785, -142.762, 65.137, 163.25] to (-231.16, 137.42, -44.5) mm, rotated rx 180 ry 0 rz 0.01 deg; joints [33.148, -43.412, 102.1, -142.805, 64.8, 163.068]
  MoveC 4750 to (-239.22, 138.68, -44.5) mm, rotated rx 180 ry 0 rz 0.01 deg; joints [33.022, -43.085, 101.395, -142.829, 64.459, 162.873] to (-247.24, 140.13, -44.5) mm, rotated rx 180 ry 0 rz 0.01 deg; joints [32.904, -42.753, 100.678, -142.841, 64.114, 162.67]
  MoveC 4751 to (-248.96, 139.35, -44.5) mm, rotated rx -180 ry 0 rz 0.01 deg; joints [32.845, -42.707, 100.58, -142.888, 64.054, 162.664] to (-248.78, 137.47, -44.5) mm, rotated rx -180 ry 0 rz 0.01 deg; joints [32.79, -42.757, 100.692, -142.965, 64.086, 162.731]
  MoveC 4752 to (-243.48, 131.17, -44.5) mm, rotated rx -180 ry 0 rz 0.01 deg; joints [32.699, -43.1, 101.441, -143.178, 64.381, 163.044] to (-238.41, 124.7, -44.5) mm, rotated rx -180 ry 0 rz 0.01 deg; joints [32.596, -43.437, 102.176, -143.399, 64.669, 163.356]
  MoveC 4753 to (-233.65, 117.98, -44.5) mm, rotated rx -180 ry 0 rz 0.01 deg; joints [32.479, -43.764, 102.893, -143.632, 64.946, 163.666] to (-229.32, 110.99, -44.5) mm, rotated rx 180 ry 0 rz 0.01 deg; joints [32.342, -44.078, 103.586, -143.879, 65.21, 163.974]
  MoveC 4754 to (-228.3, 109.14, -44.5) mm, rotated rx 180 ry 0 rz 0.01 deg; joints [32.304, -44.157, 103.758, -143.946, 65.274, 164.053] to (-227.33, 107.27, -44.5) mm, rotated rx 180 ry 0 rz 0.01 deg; joints [32.263, -44.233, 103.927, -144.013, 65.337, 164.131]
  MoveC 4755 to (-226.37, 105.39, -44.5) mm, rotated rx -180 ry 0 rz 0.01 deg; joints [32.222, -44.31, 104.096, -144.081, 65.4, 164.209] to (-225.34, 103.55, -44.5) mm, rotated rx -180 ry 0 rz 0.01 deg; joints [32.183, -44.388, 104.268, -144.147, 65.464, 164.287]
  MoveC 4756 to (-222.24, 100.44, -44.5) mm, rotated rx -180 ry 0 rz 0.01 deg; joints [32.146, -44.568, 104.665, -144.244, 65.629, 164.442] to (-218, 99.3, -44.5) mm, rotated rx -180 ry 0 rz 0.01 deg; joints [32.195, -44.746, 105.052, -144.247, 65.813, 164.555]
  MoveL 4757 to (-175.52, 99.3, -44.5) mm, rotated rx -180 ry 0 rz 0.01 deg; joints [33.09, -46.244, 108.31, -143.76, 67.49, 165.301]
  MoveC 4758 to (-171.27, 100.44, -44.5) mm, rotated rx 180 ry 0 rz 0.01 deg; joints [33.219, -46.366, 108.573, -143.659, 67.64, 165.339] to (-168.16, 103.55, -44.5) mm, rotated rx -180 ry 0 rz 0.01 deg; joints [33.39, -46.406, 108.654, -143.492, 67.72, 165.296]
  MoveC 4759 to (-167.07, 105.5, -44.5) mm, rotated rx 180 ry 0 rz 0.01 deg; joints [33.478, -46.401, 108.639, -143.398, 67.737, 165.254] to (-166.05, 107.49, -44.5) mm, rotated rx -180 ry 0 rz 0.01 deg; joints [33.566, -46.393, 108.618, -143.304, 67.751, 165.21]
  MoveC 4760 to (-165.02, 109.47, -44.5) mm, rotated rx -180 ry 0 rz 0.01 deg; joints [33.654, -46.384, 108.596, -143.209, 67.764, 165.166] to (-163.94, 111.42, -44.5) mm, rotated rx -180 ry 0 rz 0.01 deg; joints [33.742, -46.379, 108.58, -143.115, 67.781, 165.124]
  MoveC 4761 to (-159.66, 118.3, -44.5) mm, rotated rx -180 ry 0 rz 0.01 deg; joints [34.063, -46.373, 108.555, -142.778, 67.855, 164.982] to (-154.95, 124.9, -44.5) mm, rotated rx -180 ry 0 rz 0.01 deg; joints [34.383, -46.387, 108.572, -142.447, 67.949, 164.856]
  MoveC 4762 to (-149.93, 131.26, -44.5) mm, rotated rx 180 ry 0 rz 0.01 deg; joints [34.703, -46.414, 108.619, -142.121, 68.056, 164.742] to (-144.73, 137.47, -44.5) mm, rotated rx -180 ry 0 rz 0.01 deg; joints [35.023, -46.45, 108.685, -141.799, 68.172, 164.636]
  MoveC 4763 to (-144.55, 139.35, -44.5) mm, rotated rx 180 ry 0 rz 0.01 deg; joints [35.088, -46.413, 108.602, -141.72, 68.154, 164.579] to (-146.27, 140.13, -44.5) mm, rotated rx -180 ry 0 rz 0.01 deg; joints [35.074, -46.337, 108.435, -141.712, 68.078, 164.523]
  MoveC 4764 to (-163.3, 137.6, -44.5) mm, rotated rx -180 ry 0 rz 0.01 deg; joints [34.609, -45.816, 107.304, -142.038, 67.463, 164.303] to (-180.49, 136.55, -44.5) mm, rotated rx -180 ry 0 rz 0.01 deg; joints [34.196, -45.246, 106.066, -142.294, 66.813, 164.03]
  MoveL 4765 to (-203.77, 136.28, -44.5) mm, rotated rx -180 ry 0 rz 0.01 deg; joints [33.686, -44.43, 104.3, -142.571, 65.906, 163.616]
  MoveC 4766 to (-206.84, 137.2, -44.5) mm, rotated rx 180 ry 0 rz 0.01 deg; joints [33.65, -44.3, 104.015, -142.566, 65.773, 163.529] to (-208.87, 139.67, -44.5) mm, rotated rx -180 ry 0 rz 0.01 deg; joints [33.686, -44.17, 103.73, -142.487, 65.661, 163.41]
  MoveC 4767 to (-210.91, 142.14, -44.5) mm, rotated rx 180 ry 0 rz 0.01 deg; joints [33.721, -44.039, 103.444, -142.407, 65.548, 163.29] to (-213.97, 143.06, -44.5) mm, rotated rx -180 ry 0 rz 0.01 deg; joints [33.685, -43.908, 103.158, -142.401, 65.415, 163.202]
  MoveL 4768 to (-214.9, 143.06, -44.5) mm, rotated rx 180 ry 0 rz 0.01 deg; joints [33.666, -43.874, 103.086, -142.411, 65.378, 163.185]
  MoveC 4769 to (-230.28, 143.9, -44.5) mm, rotated rx 180 ry 0 rz 0.01 deg; joints [33.371, -43.294, 101.834, -142.529, 64.753, 162.867] to (-245.47, 146.39, -44.5) mm, rotated rx 180 ry 0 rz 0.01 deg; joints [33.137, -42.672, 100.493, -142.566, 64.107, 162.491]
  MoveC 4770 to (-260.34, 150.38, -44.5) mm, rotated rx -180 ry 0 rz 0.01 deg; joints [32.959, -42.017, 99.082, -142.526, 63.448, 162.063] to (-274.8, 155.69, -44.5) mm, rotated rx 180 ry 0 rz 0.01 deg; joints [32.835, -41.336, 97.616, -142.416, 62.784, 161.588]
  MoveC 4771 to (-276.35, 155.16, -44.5) mm, rotated rx -180 ry 0 rz 0.01 deg; joints [32.787, -41.289, 97.515, -142.449, 62.726, 161.575] to (-276.02, 153.55, -44.5) mm, rotated rx 180 ry 0 rz 0.01 deg; joints [32.744, -41.34, 97.628, -142.514, 62.76, 161.638]
  MoveC 4772 to (-267.11, 146.3, -44.5) mm, rotated rx -180 ry 0 rz 0.01 deg; joints [32.697, -41.856, 98.744, -142.749, 63.221, 162.07] to (-258.77, 138.4, -44.5) mm, rotated rx 180 ry 0 rz 0.01 deg; joints [32.618, -42.359, 99.836, -143.011, 63.665, 162.506]
  MoveC 4773 to (-251, 129.94, -44.5) mm, rotated rx 180 ry 0 rz 0.01 deg; joints [32.508, -42.848, 100.901, -143.296, 64.09, 162.942] to (-243.78, 121, -44.5) mm, rotated rx 180 ry 0 rz 0.01 deg; joints [32.37, -43.321, 101.935, -143.602, 64.497, 163.378]
  MoveC 4774 to (-241.44, 117.78, -44.5) mm, rotated rx -180 ry 0 rz 0.01 deg; joints [32.314, -43.481, 102.284, -143.714, 64.633, 163.528] to (-239.24, 114.46, -44.5) mm, rotated rx 180 ry 0 rz 0.01 deg; joints [32.253, -43.637, 102.626, -143.831, 64.765, 163.678]
  MoveC 4775 to (-237.14, 111.08, -44.5) mm, rotated rx 180 ry 0 rz 0.01 deg; joints [32.186, -43.79, 102.962, -143.952, 64.893, 163.828] to (-235.12, 107.65, -44.5) mm, rotated rx 180 ry 0 rz 0.01 deg; joints [32.117, -43.94, 103.294, -144.074, 65.018, 163.977]
  MoveC 4776 to (-233.62, 104.94, -44.5) mm, rotated rx -180 ry 0 rz 0.01 deg; joints [32.06, -44.055, 103.547, -144.172, 65.113, 164.092] to (-232.2, 102.19, -44.5) mm, rotated rx 180 ry 0 rz 0.01 deg; joints [32, -44.168, 103.795, -144.272, 65.205, 164.206]
  MoveC 4777 to (-230.78, 99.45, -44.5) mm, rotated rx 180 ry 0 rz 0.01 deg; joints [31.939, -44.28, 104.042, -144.372, 65.297, 164.32] to (-229.28, 96.74, -44.5) mm, rotated rx 180 ry 0 rz 0.01 deg; joints [31.882, -44.393, 104.293, -144.469, 65.392, 164.434]
  MoveC 4778 to (-226.17, 93.63, -44.5) mm, rotated rx 180 ry 0 rz 0.01 deg; joints [31.843, -44.574, 104.689, -144.567, 65.557, 164.589] to (-221.93, 92.49, -44.5) mm, rotated rx -180 ry 0 rz 0.01 deg; joints [31.892, -44.752, 105.077, -144.57, 65.742, 164.701]
  MoveL 4779 to (-171.59, 92.49, -44.5) mm, rotated rx 180 ry 0 rz 0.01 deg; joints [32.948, -46.526, 108.938, -143.991, 67.731, 165.58]
  MoveC 4780 to (-167.34, 93.63, -44.5) mm, rotated rx 180 ry 0 rz 0.01 deg; joints [33.078, -46.647, 109.201, -143.89, 67.881, 165.618] to (-164.23, 96.74, -44.5) mm, rotated rx -180 ry 0 rz 0.01 deg; joints [33.25, -46.687, 109.282, -143.722, 67.961, 165.575]
  MoveC 4781 to (-162.67, 99.55, -44.5) mm, rotated rx -180 ry 0 rz 0.01 deg; joints [33.377, -46.68, 109.261, -143.586, 67.985, 165.515] to (-161.19, 102.41, -44.5) mm, rotated rx -180 ry 0 rz 0.01 deg; joints [33.504, -46.669, 109.231, -143.449, 68.004, 165.452]
  MoveC 4782 to (-159.71, 105.27, -44.5) mm, rotated rx 180 ry 0 rz 0.01 deg; joints [33.632, -46.657, 109.2, -143.313, 68.024, 165.389] to (-158.15, 108.08, -44.5) mm, rotated rx -180 ry 0 rz 0.01 deg; joints [33.759, -46.649, 109.177, -143.177, 68.047, 165.329]
  MoveC 4783 to (-149.76, 120.95, -44.5) mm, rotated rx -180 ry 0 rz 0.01 deg; joints [34.37, -46.65, 109.155, -142.539, 68.199, 165.071] to (-140.05, 132.86, -44.5) mm, rotated rx -180 ry 0 rz 0.01 deg; joints [34.98, -46.711, 109.264, -141.922, 68.409, 164.864]
  MoveC 4784 to (-129.22, 143.74, -44.5) mm, rotated rx -180 ry 0 rz 0.01 deg; joints [35.583, -46.825, 109.493, -141.329, 68.672, 164.707] to (-117.43, 153.59, -44.5) mm, rotated rx 180 ry 0 rz 0.01 deg; joints [36.177, -46.987, 109.83, -140.761, 68.979, 164.598]
  MoveC 4785 to (-117.11, 155.2, -44.5) mm, rotated rx 180 ry 0 rz 0.01 deg; joints [36.237, -46.961, 109.769, -140.691, 68.969, 164.552] to (-118.67, 155.72, -44.5) mm, rotated rx 180 ry 0 rz 0.01 deg; joints [36.217, -46.898, 109.63, -140.694, 68.905, 164.508]
  MoveC 4786 to (-129.21, 151.68, -44.5) mm, rotated rx 180 ry 0 rz 0.01 deg; joints [35.84, -46.643, 109.081, -141.008, 68.567, 164.453] to (-140.02, 148.43, -44.5) mm, rotated rx 180 ry 0 rz 0.01 deg; joints [35.485, -46.358, 108.463, -141.29, 68.204, 164.367]
  MoveC 4787 to (-151.02, 145.93, -44.5) mm, rotated rx -180 ry 0 rz 0.01 deg; joints [35.154, -46.044, 107.785, -141.54, 67.822, 164.253] to (-162.16, 144.13, -44.5) mm, rotated rx -180 ry 0 rz 0.01 deg; joints [34.845, -45.706, 107.052, -141.758, 67.421, 164.113]
  MoveC 4788 to (-170.37, 143.33, -44.5) mm, rotated rx -180 ry 0 rz 0.01 deg; joints [34.636, -45.442, 106.479, -141.894, 67.116, 163.992] to (-178.62, 143.06, -44.5) mm, rotated rx -180 ry 0 rz 0.01 deg; joints [34.446, -45.162, 105.872, -142.005, 66.801, 163.852]
  MoveL 4789 to (-213.97, 143.06, -44.5) mm, rotated rx 180 ry 0 rz 0.01 deg; joints [33.685, -43.908, 103.158, -142.401, 65.415, 163.202]
  MoveC 4790 to (-217.01, 143.99, -44.5) mm, rotated rx -180 ry 0 rz 0.01 deg; joints [33.651, -43.776, 102.873, -142.394, 65.282, 163.115] to (-219.01, 146.45, -44.5) mm, rotated rx 180 ry 0 rz 0.01 deg; joints [33.686, -43.646, 102.588, -142.313, 65.171, 162.994]
  MoveC 4791 to (-220.97, 148.94, -44.5) mm, rotated rx -180 ry 0 rz 0.01 deg; joints [33.724, -43.517, 102.305, -142.231, 65.061, 162.874] to (-223.94, 150.01, -44.5) mm, rotated rx 180 ry 0 rz 0.01 deg; joints [33.695, -43.383, 102.015, -142.216, 64.929, 162.781]
  MoveC 4792 to (-237.13, 151.53, -44.5) mm, rotated rx 180 ry 0 rz 0.01 deg; joints [33.468, -42.862, 100.891, -142.279, 64.379, 162.477] to (-250.12, 154.32, -44.5) mm, rotated rx -180 ry 0 rz 0.01 deg; joints [33.289, -42.31, 99.703, -142.278, 63.817, 162.129]
  MoveC 4793 to (-267.04, 159.79, -44.5) mm, rotated rx 180 ry 0 rz 0.01 deg; joints [33.116, -41.536, 98.036, -142.187, 63.053, 161.601] to (-283.29, 167.01, -44.5) mm, rotated rx -180 ry 0 rz 0.01 deg; joints [33.013, -40.73, 96.303, -142.002, 62.287, 161.011]
  MoveC 4794 to (-285.56, 166.92, -44.5) mm, rotated rx 180 ry 0 rz 0.01 deg; joints [32.965, -40.643, 96.119, -142.021, 62.193, 160.967] to (-286.67, 164.94, -44.5) mm, rotated rx -180 ry 0 rz 0.01 deg; joints [32.883, -40.648, 96.133, -142.111, 62.172, 161.015]
  MoveL 4795 to (-286.67, 156.53, -44.5) mm, rotated rx 180 ry 0 rz 0.01 deg; joints [32.626, -40.853, 96.585, -142.463, 62.278, 161.315]
  MoveC 4796 to (-285.89, 153.38, -44.5) mm, rotated rx 180 ry 0 rz 0.01 deg; joints [32.544, -40.96, 96.817, -142.59, 62.35, 161.443] to (-283.75, 150.94, -44.5) mm, rotated rx 180 ry 0 rz 0.01 deg; joints [32.512, -41.103, 97.126, -142.677, 62.471, 161.573]
  MoveC 4797 to (-274.06, 143.55, -44.5) mm, rotated rx 180 ry 0 rz 0.01 deg; joints [32.474, -41.654, 98.317, -142.916, 62.968, 162.027] to (-265.07, 135.34, -44.5) mm, rotated rx 180 ry 0 rz 0.01 deg; joints [32.396, -42.191, 99.482, -143.189, 63.444, 162.487]
  MoveC 4798 to (-256.76, 126.44, -44.5) mm, rotated rx 180 ry 0 rz 0.01 deg; joints [32.282, -42.712, 100.615, -143.491, 63.898, 162.95] to (-249.08, 116.99, -44.5) mm, rotated rx 180 ry 0 rz 0.01 deg; joints [32.135, -43.215, 101.712, -143.817, 64.332, 163.411]
  MoveC 4799 to (-244.72, 110.83, -44.5) mm, rotated rx 180 ry 0 rz 0.01 deg; joints [32.026, -43.515, 102.371, -144.033, 64.587, 163.696] to (-240.77, 104.39, -44.5) mm, rotated rx 180 ry 0 rz 0.01 deg; joints [31.898, -43.804, 103.006, -144.264, 64.829, 163.979]
  MoveC 4800 to (-238.8, 100.85, -44.5) mm, rotated rx 180 ry 0 rz 0.01 deg; joints [31.823, -43.955, 103.337, -144.392, 64.954, 164.13] to (-236.95, 97.24, -44.5) mm, rotated rx 180 ry 0 rz 0.01 deg; joints [31.743, -44.102, 103.662, -144.524, 65.075, 164.28]
  MoveC 4801 to (-235.09, 93.64, -44.5) mm, rotated rx -180 ry 0 rz 0.01 deg; joints [31.663, -44.248, 103.985, -144.656, 65.196, 164.429] to (-233.12, 90.09, -44.5) mm, rotated rx -180 ry 0 rz 0.01 deg; joints [31.587, -44.397, 104.313, -144.784, 65.32, 164.577]
  MoveC 4802 to (-230.02, 86.99, -44.5) mm, rotated rx 180 ry 0 rz 0.01 deg; joints [31.548, -44.577, 104.709, -144.882, 65.485, 164.732] to (-225.77, 85.85, -44.5) mm, rotated rx 180 ry 0 rz 0.01 deg; joints [31.596, -44.756, 105.098, -144.886, 65.671, 164.843]
  MoveL 4803 to (-167.76, 85.85, -44.5) mm, rotated rx 180 ry 0 rz 0.01 deg; joints [32.809, -46.798, 109.547, -144.216, 67.966, 165.849]
  MoveC 4804 to (-163.51, 86.99, -44.5) mm, rotated rx -180 ry 0 rz 0.01 deg; joints [32.939, -46.919, 109.81, -144.114, 68.116, 165.887] to (-160.4, 90.09, -44.5) mm, rotated rx -180 ry 0 rz 0.01 deg; joints [33.111, -46.959, 109.891, -143.945, 68.196, 165.845]
  MoveC 4805 to (-158.36, 93.74, -44.5) mm, rotated rx 180 ry 0 rz 0.01 deg; joints [33.278, -46.951, 109.865, -143.768, 68.227, 165.768] to (-156.45, 97.45, -44.5) mm, rotated rx 180 ry 0 rz 0.01 deg; joints [33.444, -46.936, 109.827, -143.59, 68.252, 165.686]
  MoveC 4806 to (-154.53, 101.16, -44.5) mm, rotated rx 180 ry 0 rz 0.01 deg; joints [33.61, -46.922, 109.787, -143.412, 68.277, 165.605] to (-152.49, 104.81, -44.5) mm, rotated rx -180 ry 0 rz 0.01 deg; joints [33.776, -46.912, 109.758, -143.236, 68.307, 165.527]
  MoveC 4807 to (-143.79, 118.06, -44.5) mm, rotated rx 180 ry 0 rz 0.01 deg; joints [34.409, -46.915, 109.74, -142.576, 68.464, 165.265] to (-133.63, 130.23, -44.5) mm, rotated rx -180 ry 0 rz 0.01 deg; joints [35.04, -46.984, 109.867, -141.939, 68.686, 165.059]
  MoveC 4808 to (-122.22, 141.22, -44.5) mm, rotated rx -180 ry 0 rz 0.01 deg; joints [35.664, -47.113, 110.13, -141.33, 68.967, 164.909] to (-109.74, 150.98, -44.5) mm, rotated rx -180 ry 0 rz 0.01 deg; joints [36.275, -47.298, 110.517, -140.751, 69.298, 164.816]
  MoveC 4809 to (-107.61, 153.42, -44.5) mm, rotated rx 180 ry 0 rz 0.01 deg; joints [36.405, -47.312, 110.542, -140.621, 69.343, 164.775] to (-106.84, 156.56, -44.5) mm, rotated rx 180 ry 0 rz 0.01 deg; joints [36.524, -47.264, 110.431, -140.484, 69.329, 164.688]
  MoveL 4810 to (-106.84, 164.94, -44.5) mm, rotated rx 180 ry 0 rz 0.01 deg; joints [36.794, -47.069, 109.988, -140.148, 69.217, 164.418]
  MoveC 4811 to (-107.95, 166.92, -44.5) mm, rotated rx 180 ry 0 rz 0.01 deg; joints [36.831, -46.987, 109.804, -140.085, 69.149, 164.334] to (-110.22, 167.01, -44.5) mm, rotated rx -180 ry 0 rz 0.01 deg; joints [36.779, -46.911, 109.638, -140.116, 69.065, 164.291]
  MoveC 4812 to (-116.14, 164.08, -44.5) mm, rotated rx 180 ry 0 rz 0.01 deg; joints [36.545, -46.786, 109.37, -140.321, 68.886, 164.282] to (-122.11, 161.28, -44.5) mm, rotated rx 180 ry 0 rz 0.01 deg; joints [36.314, -46.655, 109.089, -140.52, 68.703, 164.268]
  MoveC 4813 to (-128.19, 158.71, -44.5) mm, rotated rx -180 ry 0 rz 0.01 deg; joints [36.089, -46.514, 108.785, -140.711, 68.511, 164.244] to (-134.41, 156.5, -44.5) mm, rotated rx 180 ry 0 rz 0.01 deg; joints [35.873, -46.358, 108.45, -140.887, 68.308, 164.205]
  MoveC 4814 to (-154.15, 151.71, -44.5) mm, rotated rx -180 ry 0 rz 0.01 deg; joints [35.268, -45.804, 107.252, -141.347, 67.626, 164.009] to (-174.39, 149.94, -44.5) mm, rotated rx 180 ry 0 rz 0.01 deg; joints [34.759, -45.15, 105.833, -141.674, 66.875, 163.703]
  MoveL 4815 to (-214.9, 149.71, -44.5) mm, rotated rx -180 ry 0 rz 0.01 deg; joints [33.876, -43.719, 102.74, -142.138, 65.293, 162.963]
  MoveC 4816 to (-219.42, 149.78, -44.5) mm, rotated rx -180 ry 0 rz 0.01 deg; joints [33.783, -43.553, 102.382, -142.181, 65.112, 162.875] to (-223.94, 150.01, -44.5) mm, rotated rx -180 ry 0 rz 0.01 deg; joints [33.695, -43.383, 102.015, -142.216, 64.929, 162.781]
  MoveC 4817 to (-227.57, 151.39, -44.5) mm, rotated rx 180 ry 0 rz 0.01 deg; joints [33.662, -43.217, 101.656, -142.195, 64.765, 162.665] to (-229.81, 154.57, -44.5) mm, rotated rx 180 ry 0 rz 0.01 deg; joints [33.715, -43.06, 101.312, -142.085, 64.635, 162.514]
  MoveC 4818 to (-231.97, 157.78, -44.5) mm, rotated rx -180 ry 0 rz 0.01 deg; joints [33.771, -42.904, 100.972, -141.973, 64.507, 162.363] to (-235.49, 159.38, -44.5) mm, rotated rx 180 ry 0 rz 0.01 deg; joints [33.747, -42.736, 100.607, -141.94, 64.345, 162.24]
  MoveC 4819 to (-264.73, 167.21, -44.5) mm, rotated rx -180 ry 0 rz 0.01 deg; joints [33.39, -41.444, 97.827, -141.861, 63.054, 161.386] to (-291.54, 181.27, -44.5) mm, rotated rx -180 ry 0 rz 0.01 deg; joints [33.281, -40.05, 94.831, -141.457, 61.76, 160.319]
  MoveC 4820 to (-293.68, 181.38, -44.5) mm, rotated rx 180 ry 0 rz 0.01 deg; joints [33.242, -39.962, 94.644, -141.465, 61.668, 160.269] to (-294.79, 179.54, -44.5) mm, rotated rx 180 ry 0 rz 0.01 deg; joints [33.165, -39.964, 94.652, -141.549, 61.645, 160.313]
  MoveL 4821 to (-294.79, 153.84, -44.5) mm, rotated rx 180 ry 0 rz 0.01 deg; joints [32.385, -40.599, 96.047, -142.628, 61.97, 161.242]
  MoveC 4822 to (-293.67, 149.3, -44.5) mm, rotated rx 180 ry 0 rz 0.01 deg; joints [32.268, -40.753, 96.382, -142.811, 62.074, 161.427] to (-290.58, 145.8, -44.5) mm, rotated rx 180 ry 0 rz 0.01 deg; joints [32.22, -40.958, 96.826, -142.938, 62.249, 161.614]
  MoveC 4823 to (-282.14, 139.59, -44.5) mm, rotated rx 180 ry 0 rz 0.01 deg; joints [32.192, -41.435, 97.856, -143.14, 62.681, 162.003] to (-274.04, 132.93, -44.5) mm, rotated rx -180 ry 0 rz 0.01 deg; joints [32.143, -41.904, 98.871, -143.359, 63.102, 162.394]
  MoveC 4824 to (-266.49, 125.64, -44.5) mm, rotated rx -180 ry 0 rz 0.01 deg; joints [32.063, -42.362, 99.864, -143.604, 63.507, 162.789] to (-259.74, 117.62, -44.5) mm, rotated rx 180 ry 0 rz 0.01 deg; joints [31.943, -42.801, 100.821, -143.883, 63.887, 163.189]
  MoveC 4825 to (-256.59, 113.41, -44.5) mm, rotated rx 180 ry 0 rz 0.01 deg; joints [31.872, -43.014, 101.288, -144.032, 64.069, 163.388] to (-253.49, 109.17, -44.5) mm, rotated rx -180 ry 0 rz 0.01 deg; joints [31.798, -43.226, 101.75, -144.181, 64.25, 163.587]
  MoveC 4826 to (-250.52, 104.84, -44.5) mm, rotated rx -180 ry 0 rz 0.01 deg; joints [31.718, -43.433, 102.204, -144.335, 64.426, 163.784] to (-247.78, 100.35, -44.5) mm, rotated rx -180 ry 0 rz 0.01 deg; joints [31.628, -43.634, 102.646, -144.497, 64.594, 163.981]
  MoveC 4827 to (-245.23, 95.79, -44.5) mm, rotated rx 180 ry 0 rz 0.01 deg; joints [31.531, -43.828, 103.074, -144.663, 64.756, 164.176] to (-242.8, 91.16, -44.5) mm, rotated rx 180 ry 0 rz 0.01 deg; joints [31.429, -44.019, 103.494, -144.833, 64.913, 164.369]
  MoveC 4828 to (-240.36, 86.54, -44.5) mm, rotated rx 180 ry 0 rz 0.01 deg; joints [31.326, -44.208, 103.911, -145.002, 65.07, 164.561] to (-237.81, 81.97, -44.5) mm, rotated rx 180 ry 0 rz 0.01 deg; joints [31.228, -44.399, 104.334, -145.168, 65.232, 164.751]
  MoveC 4829 to (-234.71, 78.86, -44.5) mm, rotated rx -180 ry 0 rz 0.01 deg; joints [31.188, -44.579, 104.729, -145.267, 65.397, 164.905] to (-230.47, 77.73, -44.5) mm, rotated rx -180 ry 0 rz 0.01 deg; joints [31.235, -44.758, 105.118, -145.272, 65.583, 165.015]
  MoveL 4830 to (-163.07, 77.73, -44.5) mm, rotated rx 180 ry 0 rz 0.01 deg; joints [32.637, -47.128, 110.287, -144.49, 68.254, 166.175]
  MoveC 4831 to (-158.82, 78.86, -44.5) mm, rotated rx -180 ry 0 rz 0.01 deg; joints [32.768, -47.249, 110.549, -144.387, 68.403, 166.212] to (-155.71, 81.97, -44.5) mm, rotated rx 180 ry 0 rz 0.01 deg; joints [32.941, -47.289, 110.631, -144.218, 68.483, 166.17]
  MoveC 4832 to (-153.09, 86.64, -44.5) mm, rotated rx 180 ry 0 rz 0.01 deg; joints [33.155, -47.28, 110.601, -143.99, 68.522, 166.073] to (-150.6, 91.37, -44.5) mm, rotated rx -180 ry 0 rz 0.01 deg; joints [33.369, -47.264, 110.556, -143.762, 68.556, 165.972]
  MoveC 4833 to (-148.1, 96.09, -44.5) mm, rotated rx -180 ry 0 rz 0.01 deg; joints [33.583, -47.247, 110.51, -143.534, 68.589, 165.87] to (-145.48, 100.76, -44.5) mm, rotated rx 180 ry 0 rz 0.01 deg; joints [33.798, -47.235, 110.475, -143.306, 68.628, 165.772]
  MoveC 4834 to (-136.89, 113.78, -44.5) mm, rotated rx 180 ry 0 rz 0.01 deg; joints [34.424, -47.239, 110.459, -142.654, 68.782, 165.517] to (-126.81, 125.7, -44.5) mm, rotated rx 180 ry 0 rz 0.01 deg; joints [35.049, -47.31, 110.592, -142.025, 69.002, 165.319]
  MoveC 4835 to (-115.45, 136.39, -44.5) mm, rotated rx -180 ry 0 rz 0.01 deg; joints [35.665, -47.444, 110.865, -141.425, 69.283, 165.179] to (-102.98, 145.77, -44.5) mm, rotated rx 180 ry 0 rz 0.01 deg; joints [36.267, -47.637, 111.27, -140.858, 69.617, 165.098]
  MoveC 4836 to (-99.85, 149.23, -44.5) mm, rotated rx -180 ry 0 rz 0.01 deg; joints [36.454, -47.659, 111.311, -140.67, 69.684, 165.043] to (-98.72, 153.75, -44.5) mm, rotated rx -180 ry 0 rz 0.01 deg; joints [36.628, -47.591, 111.155, -140.471, 69.665, 164.918]
  MoveL 4837 to (-98.72, 179.54, -44.5) mm, rotated rx -180 ry 0 rz 0.01 deg; joints [37.455, -46.987, 109.782, -139.441, 69.316, 164.085]
  MoveC 4838 to (-99.83, 181.38, -44.5) mm, rotated rx -180 ry 0 rz 0.01 deg; joints [37.487, -46.907, 109.604, -139.385, 69.251, 164.005] to (-101.97, 181.27, -44.5) mm, rotated rx -180 ry 0 rz 0.01 deg; joints [37.431, -46.841, 109.458, -139.422, 69.175, 163.971]
  MoveC 4839 to (-116.36, 172.87, -44.5) mm, rotated rx 180 ry 0 rz 0.01 deg; joints [36.82, -46.572, 108.886, -139.972, 68.76, 163.992] to (-131.71, 166.4, -44.5) mm, rotated rx -180 ry 0 rz 0.01 deg; joints [36.253, -46.217, 108.124, -140.451, 68.277, 163.931]
  MoveC 4840 to (-147.69, 161.76, -44.5) mm, rotated rx -180 ry 0 rz 0.01 deg; joints [35.736, -45.79, 107.201, -140.856, 67.739, 163.797] to (-164.06, 158.77, -44.5) mm, rotated rx -180 ry 0 rz 0.01 deg; joints [35.27, -45.301, 106.145, -141.188, 67.156, 163.6]
  MoveC 4841 to (-171.32, 158.06, -44.5) mm, rotated rx 180 ry 0 rz 0.01 deg; joints [35.085, -45.067, 105.638, -141.307, 66.887, 163.491] to (-178.62, 157.83, -44.5) mm, rotated rx -180 ry 0 rz 0.01 deg; joints [34.916, -44.819, 105.101, -141.404, 66.609, 163.365]
  MoveL 4842 to (-214.9, 157.83, -44.5) mm, rotated rx -180 ry 0 rz 0.01 deg; joints [34.131, -43.528, 102.313, -141.805, 65.188, 162.688]
  MoveC 4843 to (-225.22, 158.22, -44.5) mm, rotated rx -180 ry 0 rz 0.01 deg; joints [33.925, -43.142, 101.482, -141.891, 64.772, 162.478] to (-235.49, 159.38, -44.5) mm, rotated rx -180 ry 0 rz 0.01 deg; joints [33.747, -42.736, 100.607, -141.94, 64.345, 162.24]
  MoveC 4844 to (-238.87, 161.02, -44.5) mm, rotated rx -180 ry 0 rz 0.01 deg; joints [33.728, -42.571, 100.25, -141.903, 64.188, 162.118] to (-240.75, 164.27, -44.5) mm, rotated rx 180 ry 0 rz 0.01 deg; joints [33.79, -42.422, 99.926, -141.786, 64.07, 161.968]
  MoveC 4845 to (-242.54, 167.55, -44.5) mm, rotated rx -180 ry 0 rz 0.01 deg; joints [33.854, -42.276, 99.607, -141.667, 63.956, 161.819] to (-245.78, 169.4, -44.5) mm, rotated rx 180 ry 0 rz 0.01 deg; joints [33.844, -42.11, 99.247, -141.618, 63.801, 161.69]
  MoveC 4846 to (-260.44, 173.86, -44.5) mm, rotated rx 180 ry 0 rz 0.01 deg; joints [33.68, -41.445, 97.818, -141.553, 63.146, 161.237] to (-274.56, 179.82, -44.5) mm, rotated rx -180 ry 0 rz 0.01 deg; joints [33.576, -40.753, 96.33, -141.408, 62.487, 160.732]
  MoveC 4847 to (-281.18, 183.42, -44.5) mm, rotated rx -180 ry 0 rz 0.01 deg; joints [33.552, -40.404, 95.581, -141.302, 62.166, 160.462] to (-287.44, 187.61, -44.5) mm, rotated rx 180 ry 0 rz 0.01 deg; joints [33.553, -40.052, 94.824, -141.167, 61.851, 160.174]
  MoveC 4848 to (-293.46, 192.12, -44.5) mm, rotated rx 180 ry 0 rz 0.01 deg; joints [33.569, -39.697, 94.064, -141.013, 61.541, 159.876] to (-299.41, 196.75, -44.5) mm, rotated rx 180 ry 0 rz 0.01 deg; joints [33.589, -39.34, 93.298, -140.851, 61.231, 159.573]
